// TIA Portal project "MQTT_Demo_V14" (V14)

(* hardware
DEVICE "S7-1200 station_1"  S7-1200 Station
   slot 0: "Rack_0"  Rack  V1.0
   slot 1: "MQTT_Demo"  CPU 1214C AC/DC/Rly  6ES7 214-1BG40-0XB0  V4.2
*)

// ===== PLC "MQTT_Demo"  CPU 1214C AC/DC/Rly =====

VAR_GLOBAL   // PLC tag table "Default tag table"
   "Clock_Byte" AT %MB0 : Byte;
   "Clock_10Hz" AT %M0.0 : Bool;
   "Clock_5Hz" AT %M0.1 : Bool;
   "Clock_2.5Hz" AT %M0.2 : Bool;
   "Clock_2Hz" AT %M0.3 : Bool;
   "Clock_1.25Hz" AT %M0.4 : Bool;
   "Clock_1Hz" AT %M0.5 : Bool;
   "Clock_0.625Hz" AT %M0.6 : Bool;
   "Clock_0.5Hz" AT %M0.7 : Bool;
   "System_Byte" AT %MB1 : Byte;
   "FirstScan" AT %M1.0 : Bool;
   "DiagStatusUpdate" AT %M1.1 : Bool;
   "AlwaysTRUE" AT %M1.2 : Bool;
   "AlwaysFALSE" AT %M1.3 : Bool;
   "mwTemp" AT %MW20 : Word;
   "DI_Good" AT %I0.0 : Bool;
   "DI_Bad" AT %I0.1 : Bool;
   "DQ_Error" AT %Q0.1 : Bool;
   "DQ_Busy" AT %Q0.0 : Bool;
END_VAR

TYPE "udtError_MQTT"
   STRUCT
      ConSendErr : Bool;   // Connect send error
      ConSendTO : Bool;   // Connect send timeout
      ConAckRcvErr : Bool;   // Connack receive error
      ConAckTO : Bool;   // Connack timeout
      ConAckIncReply : Bool;   // Conack incorrect reply (header)
      ConAckIncLen : Bool;   // Conack incorrect remaining length
      ConAckUnacProt : Bool;   // Conack unacceptable protocol version (0x01)
      ConAckIdRej : Bool;   // Conack ID rejected (0x02)
      ConAckSerUn : Bool;   // Conack server unavailable (0x03)
      ConAckUserPass : Bool;   // Conack incorerct user/password (0x04)
      ConAckNotAut : Bool;   // Conack not authorized (0x05)
      ConAckUnknown : Bool;   // Conack unknow erro code (>0x05)
      PubSendErr : Bool;   // Publish send error
      PubSendTO : Bool;   // Publish send timeout
      PubAckRcvErr : Bool;   // Puback receive error
      PubAckTO : Bool;   // Puback receive timeout
      PubAckIncReply : Bool;   // Puback incorerct reply (header)
      PubAckIncLen : Bool;   // Puback incorrect remaining length
      PubAckPacketID : Bool;   // Puback incorrect Packet ID
      TcpErr : Bool;   // TCP connection failed
      TcpTO : Bool;   // TCP connection timeout
      QueueOverflow : Bool;   // Queue overlow
   END_STRUCT;
END_TYPE

DATA_BLOCK "dbMQTT_Queue"   // DB1
{ S7_Optimized_Access := 'TRUE' }
VERSION : 0.1
   VAR
      iIndexWrite : Int;   // Write index
      iIndexMax : Int;   // Max elements in the queue
      bErrorOverfill : Bool;   // Queue overfill error detected
      Element : Array[1..50] of Struct
         iStatus : Int;
         iQOS : Int;
         sTopic : String;
         sValue : String;
      END_STRUCT;
   END_VAR
BEGIN
END_DATA_BLOCK

DATA_BLOCK "fbInsMaster_IBM"   // DB2
{ S7_Optimized_Access := 'TRUE' }
VERSION : 0.1
// stored: InstanceOfName fbMaster_IBM
"fbMaster_IBM"
BEGIN
END_DATA_BLOCK

DATA_BLOCK "fbInsMaster_Adafruit"   // DB4
{ S7_Optimized_Access := 'TRUE' }
VERSION : 0.1
// stored: InstanceOfName fbMaster_Adafruit
"fbMaster_Adafruit"
BEGIN
END_DATA_BLOCK

DATA_BLOCK "dbMessages"   // DB5
{ S7_Optimized_Access := 'TRUE' }
VERSION : 0.1
   VAR
      sMessage : Array[1..50] of String;
   END_VAR
BEGIN
   sMessage[1] := 'Knock Knock. Who`s there? Ice cream! Ice cream who? Ice cream if you don`t let me in!';
   sMessage[2] := 'Knock Knock. Who`s there? Noah. Noah who? Noah way to open the door?';
   sMessage[3] := 'Knock Knock. Who`s there? Cows go. Cows go who? No, cows go moo!';
   sMessage[4] := 'Knock Knock. Who`s there? Hatch. Hatch who? Bless you and please cover your mouth next time.';
   sMessage[5] := 'Knock Knock. Who`s there? Boo. Boo who? Don`t cry, it`s just a joke.';
   sMessage[6] := 'Knock Knock. Who`s there? Venice. Venice who? Venice this door gonna open?';
   sMessage[7] := 'Knock Knock. Who`s there? Lettuce! Lettuce who? Lettuce in!';
   sMessage[8] := 'Knock Knock. Who`s there? Scold. Scold who? Scold outside-let me in!';
   sMessage[9] := 'Knock Knock. Who`s there? Needle. Needle who? Needle little help gettin` in the door.';
   sMessage[10] := 'Knock Knock. Who`s there? Nana. Nana who? Nana your business who`s there.';
   sMessage[11] := 'Knock Knock. Who`s there? Isabelle. Isabelle who? Isabelle working, or should I keep knocking?';
   sMessage[12] := 'Knock Knock. Who`s there? Claire. Claire who? Claire the way; I`m coming in!';
   sMessage[13] := 'Knock Knock. Who`s there? Ben. Ben who? Ben knocking for 20 minutes!';
   sMessage[14] := 'Knock Knock. Who`s there? Tuna! Tuna who? Tuna piano and it`ll sound better!';
   sMessage[15] := 'Knock Knock. Who`s there? Snow! Snow who? Snow use, I`ve forgotten my key again!';
END_DATA_BLOCK

// folder: System blocks/Program resources

DATA_BLOCK "dbTCON_Adafruit"   // DB3
{ S7_Optimized_Access := 'TRUE' }
AUTHOR : SIMATIC
FAMILY : MC7Plus
NAME : TCON_Prm
VERSION : 1.0
// stored: InstanceOfName TCON_Param
"TCON_Param"
BEGIN
   ID := 1;
   REM_TSAP_ID[1] := B#16#07;
   REM_TSAP_ID[2] := B#16#5B;
   REM_STADDR[1] := 52;
   REM_STADDR[2] := 70;
   REM_STADDR[3] := 203;
   REM_STADDR[4] := 194;
END_DATA_BLOCK

DATA_BLOCK "dbTCON_IBM"   // DB6
{ S7_Optimized_Access := 'TRUE' }
AUTHOR : SIMATIC
FAMILY : MC7Plus
NAME : TCON_Prm
VERSION : 1.0
// stored: InstanceOfName TCON_Param
"TCON_Param"
BEGIN
   ID := 1;
   REM_TSAP_ID[1] := B#16#07;
   REM_TSAP_ID[2] := B#16#5B;
   REM_STADDR[1] := 169;
   REM_STADDR[2] := 45;
   REM_STADDR[3] := 2;
   REM_STADDR[4] := 20;
END_DATA_BLOCK

// folder: (top level)

FUNCTION_BLOCK "fbMQTT"   // FB1, SCL
{ S7_Optimized_Access := 'FALSE' }
VERSION : 0.1
   VAR_INPUT
      iInQueueSize : Int;
      sInClientID : String;   // Client ID, 23 char max
      sInUserName : String;
      sInPassword : String;
      bInCleanSession : Bool;   // 0=Reuse prev session; 1=Discard prev sessions and start new one
      bInResetError : Bool;
   END_VAR
   VAR_OUTPUT
      bOutError : Bool;
      bOutBusy : Bool;
      bOutTCPConnected : Bool;
      bOutMQTT_Connected : Bool;
      ERROR_MQTT : "udtError_MQTT";
   END_VAR
   VAR_IN_OUT
      TCON_Param : TCON_Param;
   END_VAR
   VAR
      fbTCON : TCON;
      fbTDISCON : TDISCON;
      fbTSEND : TSEND;
      fbTRCV : TRCV;
      TON_Timeout : TON_TIME;
      byData : Array[1..1000] of Byte;   // Max: id+user+password+buffer
      bTCP_Connected : Bool;
      bMQTT_Connected : Bool;
      bPubInProgress : Bool;
      iState : Int;   // Main state machine state
      iStatePrev : Int;   // Previous state
      iSelQueueIndex : Int;   // Selected queue index
      uiSendLen : UInt;   // Sending length
      udiReceiveLen : UDInt;
      uiPacketID : UInt := 1;
   END_VAR
   VAR_TEMP
      i : Int;
      iIndex : Int;
      iLen : Int;
      byTemp : Byte;
      uiTemp : UInt;
      bStateTransition : Bool;   // Transitioning between states
   END_VAR
   VAR CONSTANT
      ciStatusDisable : Int;   // Not ready
      ciStatusReady : Int := 10;   // Ready to be send to the server
      ciStateIDLE : Int := 0;
      ciStateCon : Int := 10;   // Connect
      ciStateConSend : Int := 15;
      ciStateConAck : Int := 20;
      ciStatePub : Int := 30;   // Publish
      ciStatePubSend : Int := 35;
      ciStatePubAck : Int := 40;
      ciStateEstablishTCP : Int := 50;   // Establish TCP connection
      ciStateError : Int := 60;
      ciStateRestart : Int := 70;
   END_VAR
BEGIN
   // Main state machine - case structure
   #iStatePrev := #iState;
   CASE #iState OF
           //**********************************************************************************************************************
       #ciStateIDLE: 
           // Update max queue index
           "dbMQTT_Queue".iIndexMax := #iInQueueSize;

           // Already select element to send?
           IF #iSelQueueIndex > 0 THEN
               IF #bTCP_Connected THEN
                   IF #bMQTT_Connected THEN
                       // MQTT is conencted - just publish new message
                       #iState := #ciStatePub;
                   ELSE
                       // MQTT connection is not established - sene conn message
                       #iState := #ciStateCon;
                   END_IF;
               ELSE
                   // TCP is not connected - try to establish the connection
                   #iState := #ciStateEstablishTCP;
               END_IF;
           ELSE
               // Find element in the queue to send
               FOR #i := 1 TO "dbMQTT_Queue".iIndexMax DO
                   // Check if element is ready in the queue
                   IF ("dbMQTT_Queue".Element[#i].iStatus = #ciStatusReady) THEN
                       #iSelQueueIndex := #i;
                       EXIT;
                   END_IF;
               END_FOR;
           END_IF;

           //**********************************************************************************************************************
       #ciStateCon: // Send connect message
           ////////////////////////////////////
           // Create connect message
           ////////////////////////////////////

           //********* Configure Fixed Header ***********//
           #iIndex := 1;
           #byData[#iIndex] := 2#00010000;   // Packet type 0x1; Flags 0x0 (reserved)
           #iIndex := #iIndex + 1;

           // Calculate remaining length (see MQTT doc)
           #iLen := 12 + LEN(#sInClientID);
           IF LEN(#sInUserName) > 0 THEN
               #iLen := #iLen + LEN(#sInUserName) + 2;
           END_IF;
           IF LEN(#sInPassword) > 0 THEN
               #iLen := #iLen + LEN(#sInPassword) + 2;
           END_IF;
           REPEAT
               #byTemp := INT_TO_BYTE(#iLen MOD 128);
               #iLen := #iLen / 128;
               // if there are more data to encode, set the top bit of this byte 286
               IF #iLen > 0 THEN
                   #byTemp := #byTemp OR 128;
               END_IF;
               #byData[#iIndex] := #byTemp;
               #iIndex := #iIndex + 1;
           UNTIL #iLen <= 0 END_REPEAT;

           //********* Variable Header ***********//
           #byData[#iIndex] := 16#00;    // Length MSB
           #iIndex := #iIndex + 1;
           #byData[#iIndex] := 16#04;    // Length LSB
           #iIndex := #iIndex + 1;
           #byData[#iIndex] := CHAR_TO_BYTE('M');
           #iIndex := #iIndex + 1;
           #byData[#iIndex] := CHAR_TO_BYTE('Q');
           #iIndex := #iIndex + 1;
           #byData[#iIndex] := CHAR_TO_BYTE('T');
           #iIndex := #iIndex + 1;
           #byData[#iIndex] := CHAR_TO_BYTE('T');
           #iIndex := #iIndex + 1;
           #byData[#iIndex] := 16#04;     // Protocol level 0x04
           #iIndex := #iIndex + 1;

           // Build connect flags, ignoring will message
           #byData[#iIndex] := 16#00;
           IF LEN(#sInUserName) > 0 THEN
               #byData[#iIndex] := #byData[#iIndex] OR 2#10000000;
           END_IF;
           IF LEN(#sInPassword) > 0 THEN
               #byData[#iIndex] := #byData[#iIndex] OR 2#01000000;
           END_IF;
           IF #bInCleanSession THEN
               #byData[#iIndex] := #byData[#iIndex] OR 2#00000010;
           END_IF;
           #iIndex := #iIndex + 1;
           #byData[#iIndex] := 16#0E;  // Keepalive MSB, in seconds
           #iIndex := #iIndex + 1;
           #byData[#iIndex] := 16#10;  // Keepalive LSB, in seconds
           #iIndex := #iIndex + 1;

           // Payload - client ID
           #iLen := LEN(#sInClientID);
           #byData[#iIndex] := WORD_TO_BYTE(SHR(IN := INT_TO_WORD(#iLen), N := 8));   // String lenght MSB
           #iIndex := #iIndex + 1;
           #byData[#iIndex] := WORD_TO_BYTE(INT_TO_WORD(#iLen) AND 16#00FF);   // String lenght LSB            
           #iIndex := #iIndex + 1;
           FOR #i := 1 TO #iLen DO
               #byData[#iIndex] := CHAR_TO_BYTE(#sInClientID[#i]);
               #iIndex := #iIndex + 1;
           END_FOR;

           // Payload - User name
           IF LEN(#sInUserName) > 0 THEN
               #iLen := LEN(#sInUserName);
               #byData[#iIndex] := WORD_TO_BYTE(SHR(IN := INT_TO_WORD(#iLen), N := 8));   // String lenght MSB
               #iIndex := #iIndex + 1;
               #byData[#iIndex] := WORD_TO_BYTE(INT_TO_WORD(#iLen) AND 16#00FF);   // String lenght LSB            
               #iIndex := #iIndex + 1;
               FOR #i := 1 TO #iLen DO
                   #byData[#iIndex] := CHAR_TO_BYTE(#sInUserName[#i]);
                   #iIndex := #iIndex + 1;
               END_FOR;
           END_IF;

           // Payload - password
           IF LEN(#sInPassword) > 0 THEN
               #iLen := LEN(#sInPassword);
               #byData[#iIndex] := WORD_TO_BYTE(SHR(IN := INT_TO_WORD(#iLen), N := 8));   // String lenght MSB
               #iIndex := #iIndex + 1;
               #byData[#iIndex] := WORD_TO_BYTE(INT_TO_WORD(#iLen) AND 16#00FF);   // String lenght LSB            
               #iIndex := #iIndex + 1;
               FOR #i := 1 TO #iLen DO
                   #byData[#iIndex] := CHAR_TO_BYTE(#sInPassword[#i]);
                   #iIndex := #iIndex + 1;
               END_FOR;
           END_IF;

           //********* Send Packet ***********//
           #uiSendLen := INT_TO_UINT(#iIndex - 1);   // Update packet length
           #iState := #ciStateConSend;  // Send packet packet    

           //**********************************************************************************************************************
       #ciStateConSend:
           IF #fbTSEND.DONE THEN
               // All good. Receive conack message
               // We know exactly the conack message size
               #udiReceiveLen := 4;
               #iState := #ciStateConAck;
           ELSIF #fbTSEND.ERROR THEN
               // Sending error
               #ERROR_MQTT.ConSendErr := true;
               #iState := #ciStateError;
           ELSIF #TON_Timeout.Q THEN
               #ERROR_MQTT.ConSendTO := true;
               #iState := #ciStateError;
           END_IF;

           //**********************************************************************************************************************
       #ciStateConAck:
           IF #fbTRCV.NDR THEN
               // Parse received data
               // We know that we got an expected length
               // Header should be 0x20
               IF #byData[1] <> 16#20 THEN
                   #ERROR_MQTT.ConAckIncReply := true;
                   #iState := #ciStateError;
               // Remaining lenght should be 2
               ELSIF #byData[2] <> 2 THEN
                   #ERROR_MQTT.ConAckIncLen := true;
                   #iState := #ciStateError;
               // TODO: Parse SP flag?
               // Return code should be 0    
               ELSIF #byData[4] <> 0 THEN
                   // Parse error code
                   IF #byData[4] = 1 THEN
                       #ERROR_MQTT.ConAckUnacProt := TRUE;
                   ELSIF #byData[4] = 2 THEN
                       #ERROR_MQTT.ConAckIdRej := TRUE;
                   ELSIF #byData[4] = 3 THEN
                       #ERROR_MQTT.ConAckSerUn := TRUE;
                   ELSIF #byData[4] = 4 THEN
                       #ERROR_MQTT.ConAckUserPass := TRUE;
                   ELSIF #byData[4] = 5 THEN
                       #ERROR_MQTT.ConAckNotAut := TRUE;
                   ELSE
                       #ERROR_MQTT.ConAckUnknown := TRUE;
                   END_IF;
                   #iState := #ciStateError;
               ELSE
                   // All good
                   #bMQTT_Connected := true;
                   #iState := #ciStatePub;
               END_IF;
           ELSIF #fbTRCV.ERROR THEN
               // Receive error
               #ERROR_MQTT.ConAckRcvErr := true;
               #iState := #ciStateError;
           ELSIF #TON_Timeout.Q THEN
               #ERROR_MQTT.ConAckTO := true;
               #iState := #ciStateError;
           END_IF;

           //**********************************************************************************************************************
       #ciStatePub:
           ////////////////////////////////////
           // Create publish message
           ////////////////////////////////////

           //********* Configure Fixed Header ***********//
           #iIndex := 1;
           #byData[#iIndex] := 2#00110000;   // Packet type 0x3;
           IF #bPubInProgress THEN
               #byData[#iIndex] := #byData[#iIndex] OR 2#00001000; // DUP flag. Re-delivery attempt
           ELSE
               // New send attempt - Increment Packet ID
               #uiPacketID := #uiPacketID + 1;
           END_IF;
           // QoS flag, assuming 0 by default
           IF "dbMQTT_Queue".Element[#iSelQueueIndex].iQOS = 1 THEN
               #byData[#iIndex] := #byData[#iIndex] OR 2#00000010; // QoS flag
           END_IF;
           //TODO: QoS 2 is not currently implemented by adafruit
           // TODO: Ignoring retain flag for now
           #iIndex := #iIndex + 1;

           // Calculate remaining length (see MQTT doc)
           // No lenght for the payload
           #iLen := LEN("dbMQTT_Queue".Element[#iSelQueueIndex].sTopic) + 2 + LEN("dbMQTT_Queue".Element[#iSelQueueIndex].sValue);
           IF "dbMQTT_Queue".Element[#iSelQueueIndex].iQOS > 0 THEN
               // Adding packet ID for QoS 1 and 2
               #iLen := #iLen + 2;
           END_IF;
           REPEAT
               #byTemp := INT_TO_BYTE(#iLen MOD 128);
               #iLen := #iLen / 128;
               // if there are more data to encode, set the top bit of this byte 286
               IF #iLen > 0 THEN
                   #byTemp := #byTemp OR 128;
               END_IF;
               #byData[#iIndex] := #byTemp;
               #iIndex := #iIndex + 1;
           UNTIL #iLen <= 0 END_REPEAT;

           //********* Variable Header ***********//
           // Topic name
           #iLen := LEN("dbMQTT_Queue".Element[#iSelQueueIndex].sTopic);
           #byData[#iIndex] := WORD_TO_BYTE(SHR(IN:=INT_TO_WORD(#iLen), N:=8));   // String lenght MSB
           #iIndex := #iIndex + 1;
           #byData[#iIndex] := WORD_TO_BYTE(INT_TO_WORD(#iLen) AND 16#00FF);   // String lenght LSB
           #iIndex := #iIndex + 1;
           FOR #i := 1 TO #iLen DO
               #byData[#iIndex] := CHAR_TO_BYTE("dbMQTT_Queue".Element[#iSelQueueIndex].sTopic[#i]);
               #iIndex := #iIndex + 1;
           END_FOR;
           // packet ID
           IF "dbMQTT_Queue".Element[#iSelQueueIndex].iQOS > 0 THEN
               #byData[#iIndex] := WORD_TO_BYTE(SHR(IN:=UINT_TO_WORD(#uiPacketID), N:=8));   // Packet ID MSB
               #iIndex := #iIndex + 1;
               #byData[#iIndex] := WORD_TO_BYTE(UINT_TO_WORD(#uiPacketID) AND 16#00FF);   // PacketID LSB
               #iIndex := #iIndex + 1;
           END_IF;

           //********* Payload ***********//
           // The exact data format is not defined in the MQTT spec
           // Assuming strings, without string length
           // According to the spec, server should calcualte the lenght of the payload
           #iLen := LEN("dbMQTT_Queue".Element[#iSelQueueIndex].sValue);
           FOR #i := 1 TO #iLen DO
               #byData[#iIndex] := CHAR_TO_BYTE("dbMQTT_Queue".Element[#iSelQueueIndex].sValue[#i]);
               #iIndex := #iIndex + 1;
           END_FOR;

           // Send message
           #bPubInProgress := true;
           #uiSendLen := INT_TO_UINT(#iIndex - 1);   // Update packet length
           #iState := #ciStatePubSend;

           //**********************************************************************************************************************
       #ciStatePubSend:
           IF #fbTSEND.DONE THEN
               // QoS=1: Should receive puback message
               IF "dbMQTT_Queue".Element[#iSelQueueIndex].iQOS = 1 THEN
                   #udiReceiveLen := 4;    // Wes should receive exactly 4 bytes
                   #iState := #ciStatePubAck;
               ELSE
                   // QoS=0; No response from the server
                   // Remove message from the queue
                   "dbMQTT_Queue".Element[#iSelQueueIndex].iStatus := #ciStatusDisable;
                   #iSelQueueIndex := 0;
                   #bPubInProgress := false;
                   #iState := #ciStateIDLE;
               END_IF;
               // TODO: Handle QoS 2?
           ELSIF #fbTSEND.ERROR THEN
               // Send error
               #ERROR_MQTT.PubSendErr := true;
               #iState := #ciStateError;
           ELSIF #TON_Timeout.Q THEN
               #ERROR_MQTT.PubSendTO := true;
               #iState := #ciStateError;
           END_IF;

           //**********************************************************************************************************************
       #ciStatePubAck:
           IF #fbTRCV.NDR THEN
               // Parse received data
               // We know that we got an expected length
               // Header should be 0x40
               IF #byData[1] <> 16#40 THEN
                   // Wrong pub ack header
                   #ERROR_MQTT.PubAckIncReply := TRUE;
                   #iState := #ciStateError;
               // Remaining length should be 2
               ELSIF #byData[2] <> 16#02 THEN
                   // Wrong pub ack remaining lenght
                   #ERROR_MQTT.PubAckIncLen := TRUE;
                   #iState := #ciStateError;
               ELSE
                   // Variable header = message id
                   #uiTemp := WORD_TO_UINT(SHL(IN := BYTE_TO_WORD(#byData[3]), N := 8) + BYTE_TO_WORD(#byData[4]));
                   IF #uiTemp <> #uiPacketID THEN
                       // Incorerct packet ID
                       #ERROR_MQTT.PubAckPacketID := TRUE;
                       #iState := #ciStateError;
                   ELSE
                       // All good. Reset queue and restart
                       "dbMQTT_Queue".Element[#iSelQueueIndex].iStatus := #ciStatusDisable;
                       #iSelQueueIndex := 0;
                       #bPubInProgress := false;
                       #iState := #ciStateIDLE;
                   END_IF;
               END_IF;
           ELSIF #fbTRCV.ERROR THEN
               // Receive error
               #ERROR_MQTT.PubAckRcvErr := TRUE;
               #iState := #ciStateError;
           ELSIF #TON_Timeout.Q THEN
               #ERROR_MQTT.PubAckTO := true;
               #iState := #ciStateError;
           END_IF;

           //**********************************************************************************************************************        
       #ciStateEstablishTCP:
           // Wait for done or error flag
           IF #fbTCON.DONE THEN
               // TCP connection established 
               #bTCP_Connected := true;
               #bMQTT_Connected := false;
               #iState := #ciStateCon;
           ELSIF #fbTCON.ERROR THEN
               // Connection failed
               #ERROR_MQTT.TcpErr := true;
               #iState := #ciStateError;
           ELSIF #TON_Timeout.Q THEN
               #ERROR_MQTT.TcpTO := true;
               #iState := #ciStateError;
           END_IF;

           //**********************************************************************************************************************
       #ciStateError:
           // Reset TCP connection
           #bMQTT_Connected := false;
           #bTCP_Connected := false;
           IF #fbTDISCON.DONE OR #fbTDISCON.ERROR THEN
               #iState := #ciStateRestart;
           ELSIF #TON_Timeout.Q THEN
               // Already wait for timeout, just jump to idle
               #iState := #ciStateIDLE;
           END_IF;

           //**********************************************************************************************************************
       #ciStateRestart:
           // Wait before restarting after the error
           IF #TON_Timeout.Q THEN
               // Restart from IDLE
               #iState := #ciStateIDLE;
           END_IF;

           //**********************************************************************************************************************
       ELSE    // Something is not right - reset state
           #iState := #ciStateIDLE;
   END_CASE;


   //**********************************************************************************************************************
   // Reset all errors
   IF #bInResetError THEN
       #ERROR_MQTT.ConSendErr := FALSE;
       #ERROR_MQTT.ConSendTO := FALSE;
       #ERROR_MQTT.ConAckRcvErr := FALSE;
       #ERROR_MQTT.ConAckTO := FALSE;
       #ERROR_MQTT.ConAckIncReply := FALSE;
       #ERROR_MQTT.ConAckIncLen := FALSE;
       #ERROR_MQTT.ConAckUnacProt := FALSE;
       #ERROR_MQTT.ConAckIdRej := FALSE;
       #ERROR_MQTT.ConAckSerUn := FALSE;
       #ERROR_MQTT.ConAckUserPass := FALSE;
       #ERROR_MQTT.ConAckNotAut := FALSE;
       #ERROR_MQTT.ConAckUnknown := FALSE;
       #ERROR_MQTT.PubSendErr := FALSE;
       #ERROR_MQTT.PubSendTO := FALSE;
       #ERROR_MQTT.PubAckRcvErr := FALSE;
       #ERROR_MQTT.PubAckTO := FALSE;
       #ERROR_MQTT.PubAckIncReply := FALSE;
       #ERROR_MQTT.PubAckIncLen := FALSE;
       #ERROR_MQTT.PubAckPacketID := FALSE;
       #ERROR_MQTT.TcpErr := FALSE;
       #ERROR_MQTT.TcpTO := FALSE;
       #ERROR_MQTT.QueueOverflow := FALSE;
   END_IF;

   // Queue overlow error
   IF "dbMQTT_Queue".bErrorOverfill THEN
       #ERROR_MQTT.QueueOverflow := TRUE;
       "dbMQTT_Queue".bErrorOverfill := FALSE;
   END_IF;

   // Timeoout timer
   #bStateTransition := #iState <> #iStatePrev;
   #TON_Timeout(IN := ((NOT #bStateTransition) AND (#iState <> #ciStateIDLE)), PT := T#20S);

   // At least one erorr is active - set output error flag
   #bOutError :=
       #ERROR_MQTT.ConSendErr OR
       #ERROR_MQTT.ConSendTO OR
       #ERROR_MQTT.ConAckRcvErr OR
       #ERROR_MQTT.ConAckTO OR
       #ERROR_MQTT.ConAckIncReply OR
       #ERROR_MQTT.ConAckIncLen OR
       #ERROR_MQTT.ConAckUnacProt OR
       #ERROR_MQTT.ConAckIdRej OR
       #ERROR_MQTT.ConAckSerUn OR
       #ERROR_MQTT.ConAckUserPass OR
       #ERROR_MQTT.ConAckNotAut OR
       #ERROR_MQTT.ConAckUnknown OR
       #ERROR_MQTT.PubSendErr OR
       #ERROR_MQTT.PubSendTO OR
       #ERROR_MQTT.PubAckRcvErr OR
       #ERROR_MQTT.PubAckTO OR
       #ERROR_MQTT.PubAckIncReply OR
       #ERROR_MQTT.PubAckIncLen OR
       #ERROR_MQTT.PubAckPacketID OR
       #ERROR_MQTT.TcpErr OR
       #ERROR_MQTT.TcpTO OR
       #ERROR_MQTT.QueueOverflow;

   // Block is busy output flag
   #bOutBusy := (#iState <> #ciStateIDLE) AND (NOT #bOutError);

   // TCP and MQTT conencted outputs
   #bOutTCPConnected := #bTCP_Connected;
   #bOutMQTT_Connected := #bMQTT_Connected;


   //**********************************************************************************************************************
   // Communicaiton FBs
   #fbTCON(REQ:= (#iState = #ciStateEstablishTCP),
           ID:= #TCON_Param.ID,
           CONNECT:=#TCON_Param);

   #fbTDISCON(REQ:=(#iState = #ciStateError),
              ID:=#TCON_Param.ID);

   #fbTSEND(REQ := (#iState = #ciStateConSend) OR (#iState = #ciStatePubSend),
            ID := #TCON_Param.ID,
            LEN := #uiSendLen,
            DATA := #byData);

   #fbTRCV(EN_R := (#iState = #ciStateConAck) OR (#iState = #ciStatePubAck),
           ID:=#TCON_Param.ID,
           LEN:=#udiReceiveLen,
           DATA:=#byData);

   ENO := TRUE;
END_FUNCTION_BLOCK

FUNCTION_BLOCK "fbMaster_Adafruit"   // FB2, LAD
TITLE = Master FB
{ S7_Optimized_Access := 'TRUE' }
VERSION : 0.1
   VAR
      FP_PartGood : Bool;
      FP_PartBad : Bool;
      bMachineRunning : Bool;
      bOneMinutePulse : Bool;   // One shot one minute pulse
      diPartsGoodTotal : DInt;
      diPartsBadTotal : DInt;
      diPartsTotal : DInt;
      diPartsGoodMinute : DInt;
      diPartsBadMinute : DInt;
      diPartsMinute : DInt;
      rRunTimeSec : Real;
      rAvailability : Real;
      rPerformance : Real;
      rQuality : Real;
      diQuality : DInt;
      rOEE : Real;
      diOEE_Per : DInt;   // OEE in percents
      diOEE_PerAvg : DInt;   // Average OEE in percent
      iMessageIndex : Int;
      AVG_OEE : "fbRunningAverage";
      TON_OneMinute : TON_TIME;
      MQTT_Main : "fbMQTT";
      TON_ResetError : TON_TIME;
      TOF_Busy : TOF_TIME;
      TOF_MachineRunning : TOF_TIME;
      TONR_MachineRunTime : TONR_TIME;
   END_VAR
   VAR_TEMP
      rTemp : Real;
      bBusy : Bool;
      bTCP_Connected : Bool;
      bMQTT_Connected : Bool;
   END_VAR
   VAR CONSTANT
      cdiPlannedPartPerMinute : DInt := 30;   // Parts per minute rate
      crPlannedTimeSecPerMin : Real := 60.0;   // Planned time in seconds per interval (minute)
   END_VAR
   VAR_TEMP   // added for the SCL form of the ladder/FBD networks
      _w1 : Bool;
      _w2 : Bool;
   END_VAR
BEGIN

REGION Network 1: Made Good or Bad part
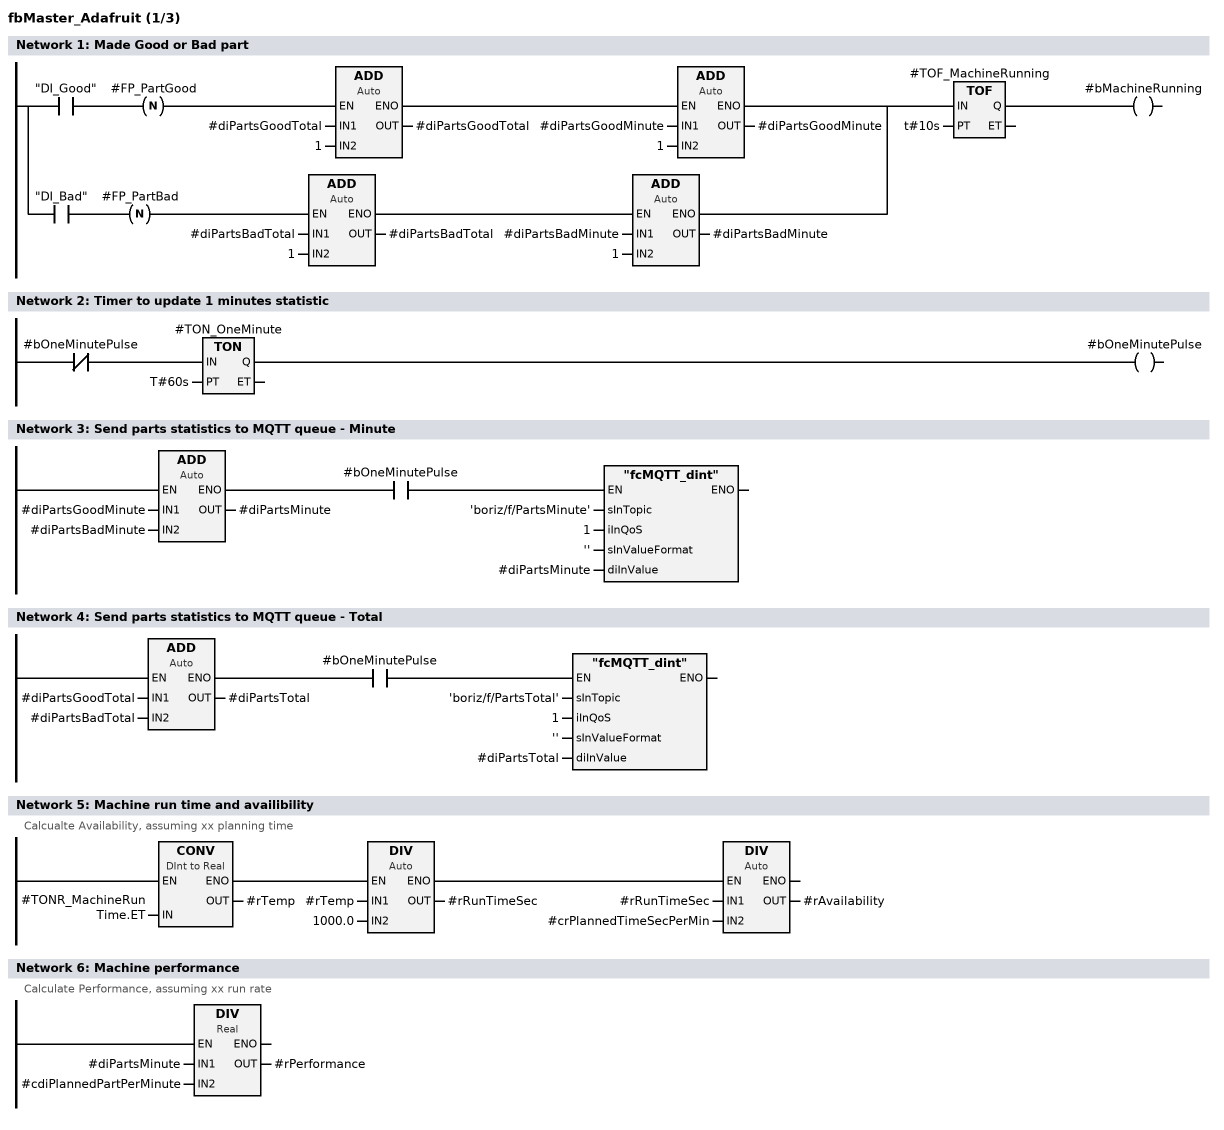
   #_w1 := NOT "DI_Good" AND #FP_PartGood;   // falling edge
   #FP_PartGood := "DI_Good";
   IF #_w1 THEN
       #diPartsGoodTotal := #diPartsGoodTotal + 1;
       #diPartsGoodMinute := #diPartsGoodMinute + 1;
   END_IF;
   #_w2 := NOT "DI_Bad" AND #FP_PartBad;   // falling edge
   #FP_PartBad := "DI_Bad";
   IF #_w2 THEN
       #diPartsBadTotal := #diPartsBadTotal + 1;
       #diPartsBadMinute := #diPartsBadMinute + 1;
   END_IF;
   #TOF_MachineRunning(IN := #_w1 OR #_w2, PT := t#10s);   // TOF
   #bMachineRunning := #TOF_MachineRunning.Q;
END_REGION

REGION Network 2: Timer to update 1 minutes statistic
   #TON_OneMinute(IN := NOT #bOneMinutePulse, PT := T#60s);   // TON
   #bOneMinutePulse := #TON_OneMinute.Q;
END_REGION

REGION Network 3: Send parts statistics to MQTT queue - Minute
   RUNG wire#powerrail
      Add(in1 := #diPartsGoodMinute, in2 := #diPartsBadMinute, out => #diPartsMinute)
      Contact( #bOneMinutePulse )
      "fcMQTT_dint"(sInTopic := 'boriz/f/PartsMinute', iInQoS := 1, sInValueFormat := '', diInValue := #diPartsMinute)
   END_RUNG
   // the same network as SCL:
   #diPartsMinute := #diPartsGoodMinute + #diPartsBadMinute;
   IF #bOneMinutePulse THEN
       "fcMQTT_dint"(sInTopic := 'boriz/f/PartsMinute',
                     iInQoS := 1,
                     sInValueFormat := '',
                     diInValue := #diPartsMinute);
   END_IF;
END_REGION

REGION Network 4: Send parts statistics to MQTT queue - Total
   RUNG wire#powerrail
      Add(in1 := #diPartsGoodTotal, in2 := #diPartsBadTotal, out => #diPartsTotal)
      Contact( #bOneMinutePulse )
      "fcMQTT_dint"(sInTopic := 'boriz/f/PartsTotal', iInQoS := 1, sInValueFormat := '', diInValue := #diPartsTotal)
   END_RUNG
   // the same network as SCL:
   #diPartsTotal := #diPartsGoodTotal + #diPartsBadTotal;
   IF #bOneMinutePulse THEN
       "fcMQTT_dint"(sInTopic := 'boriz/f/PartsTotal',
                     iInQoS := 1,
                     sInValueFormat := '',
                     diInValue := #diPartsTotal);
   END_IF;
END_REGION

REGION Network 5: Machine run time and availibility
   // Calcualte Availability, assuming xx planning time
   RUNG wire#powerrail
      { S7_Templates := "[SrcType := DInt, DestType := Real]" } Convert(in := #TONR_MachineRunTime.ET, out => #rTemp)
      Div(in1 := #rTemp, in2 := 1000.0, out => #rRunTimeSec)
      Div(in1 := #rRunTimeSec, in2 := #crPlannedTimeSecPerMin, out => #rAvailability)
   END_RUNG
   // the same network as SCL:
   #rTemp := DINT_TO_REAL(#TONR_MachineRunTime.ET);
   #rRunTimeSec := #rTemp / 1000.0;
   #rAvailability := #rRunTimeSec / #crPlannedTimeSecPerMin;
END_REGION

REGION Network 6: Machine performance
   // Calculate Performance, assuming xx run rate
   RUNG wire#powerrail
      { S7_Templates := "SrcType := Real" } Div(in1 := #diPartsMinute, in2 := #cdiPlannedPartPerMinute, out => #rPerformance)
   END_RUNG
   // the same network as SCL:
   #rPerformance := #diPartsMinute / #cdiPlannedPartPerMinute;
END_REGION

REGION Network 7: Machine quality
   // Calculate Quality
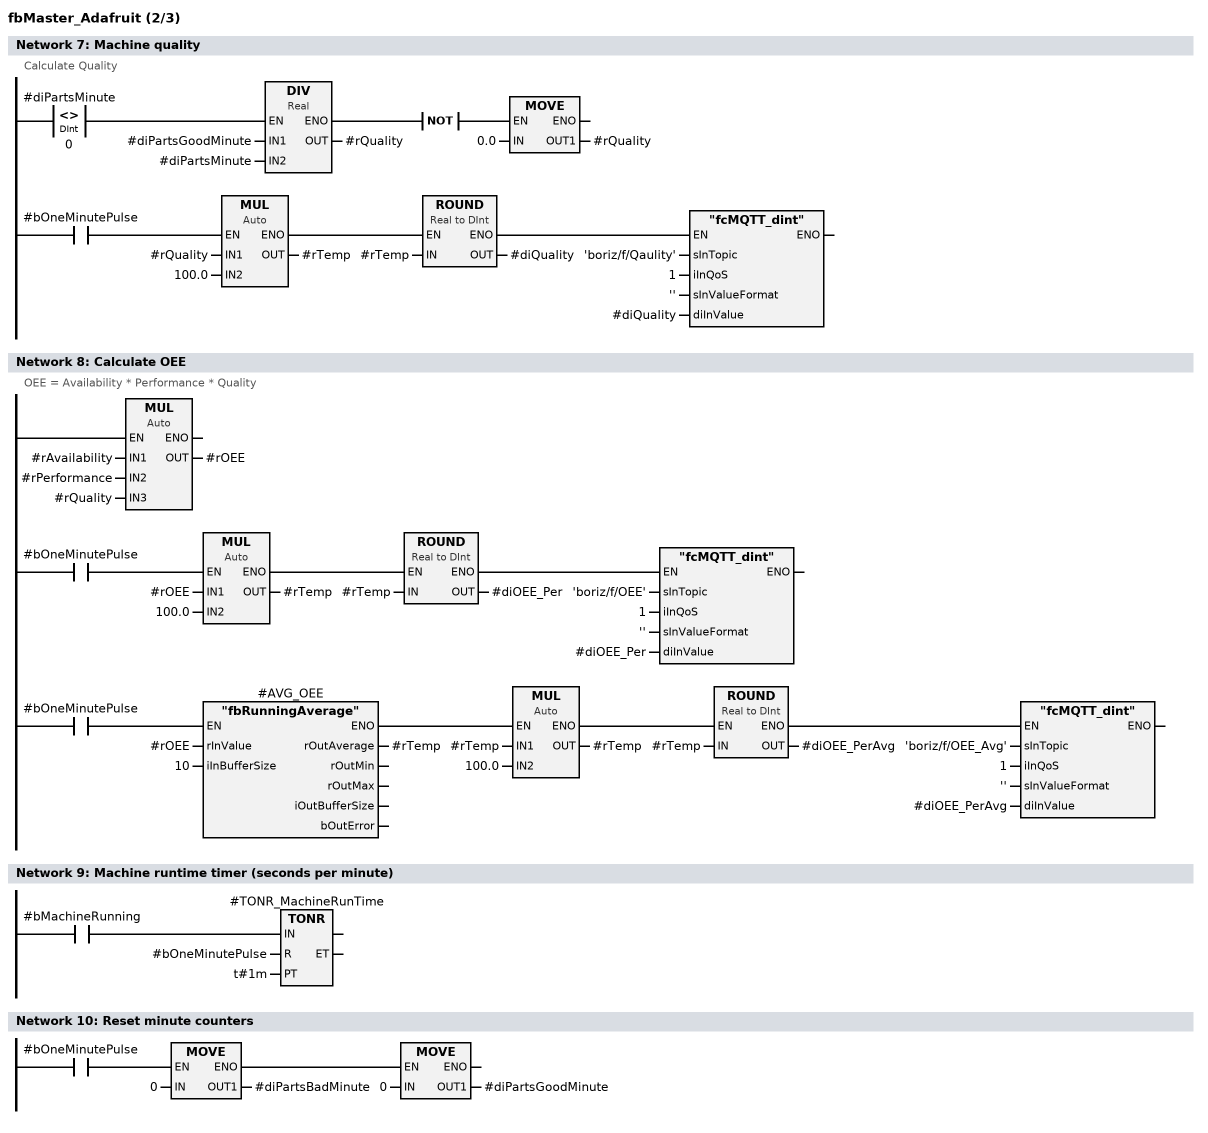
   RUNG wire#powerrail
      { S7_Templates := "SrcType := DInt" } NE_Contact(in1 := #diPartsMinute, in2 := 0)
      { S7_Templates := "SrcType := Real" } Div(in1 := #diPartsGoodMinute, in2 := #diPartsMinute, out => #rQuality)
      Not()
      Move(in := 0.0, out1 => #rQuality)
   END_RUNG
   RUNG wire#powerrail
      Contact( #bOneMinutePulse )
      Mul(in1 := #rQuality, in2 := 100.0, out => #rTemp)
      { S7_Templates := "[SrcType := Real, DestType := DInt]" } Round(in := #rTemp, out => #diQuality)
      "fcMQTT_dint"(sInTopic := 'boriz/f/Qaulity', iInQoS := 1, sInValueFormat := '', diInValue := #diQuality)
   END_RUNG
   // the same network as SCL:
   #_w1 := #diPartsMinute <> 0;
   IF #_w1 THEN #rQuality := #diPartsGoodMinute / #diPartsMinute; END_IF;
   IF NOT #_w1 THEN #rQuality := 0.0; END_IF;
   IF #bOneMinutePulse THEN
       #rTemp := #rQuality * 100.0;
       #diQuality := ROUND(#rTemp);
       "fcMQTT_dint"(sInTopic := 'boriz/f/Qaulity', iInQoS := 1, sInValueFormat := '', diInValue := #diQuality);
   END_IF;
END_REGION

REGION Network 8: Calculate OEE
   // OEE = Availability * Performance * Quality
   RUNG wire#powerrail
      Mul(in1 := #rAvailability, in2 := #rPerformance, in3 := #rQuality, out => #rOEE)
   END_RUNG
   RUNG wire#powerrail
      Contact( #bOneMinutePulse )
      Mul(in1 := #rOEE, in2 := 100.0, out => #rTemp)
      { S7_Templates := "[SrcType := Real, DestType := DInt]" } Round(in := #rTemp, out => #diOEE_Per)
      "fcMQTT_dint"(sInTopic := 'boriz/f/OEE', iInQoS := 1, sInValueFormat := '', diInValue := #diOEE_Per)
   END_RUNG
   RUNG wire#powerrail
      Contact( #bOneMinutePulse )
      #AVG_OEE(rInValue := #rOEE, iInBufferSize := 10, rOutAverage => #rTemp, rOutMin =>, rOutMax =>, iOutBufferSize =>, bOutError =>)
      Mul(in1 := #rTemp, in2 := 100.0, out => #rTemp)
      { S7_Templates := "[SrcType := Real, DestType := DInt]" } Round(in := #rTemp, out => #diOEE_PerAvg)
      "fcMQTT_dint"(sInTopic := 'boriz/f/OEE_Avg', iInQoS := 1, sInValueFormat := '', diInValue := #diOEE_PerAvg)
   END_RUNG
   // the same network as SCL:
   #rOEE := #rAvailability * #rPerformance * #rQuality;
   IF #bOneMinutePulse THEN
       #rTemp := #rOEE * 100.0;
       #diOEE_Per := ROUND(#rTemp);
       "fcMQTT_dint"(sInTopic := 'boriz/f/OEE', iInQoS := 1, sInValueFormat := '', diInValue := #diOEE_Per);
   END_IF;
   #AVG_OEE(EN := #bOneMinutePulse, rInValue := #rOEE, iInBufferSize := 10, rOutAverage => #rTemp, ENO => #_w1);   // "fbRunningAverage"
   IF #_w1 THEN
       #rTemp := #rTemp * 100.0;
       #diOEE_PerAvg := ROUND(#rTemp);
       "fcMQTT_dint"(sInTopic := 'boriz/f/OEE_Avg', iInQoS := 1, sInValueFormat := '', diInValue := #diOEE_PerAvg);
   END_IF;
END_REGION

REGION Network 9: Machine runtime timer (seconds per minute)
   #TONR_MachineRunTime(IN := #bMachineRunning, R := #bOneMinutePulse, PT := t#1m);   // TONR
END_REGION

REGION Network 10: Reset minute counters
   RUNG wire#powerrail
      Contact( #bOneMinutePulse )
      Move(in := 0, out1 => #diPartsBadMinute)
      Move(in := 0, out1 => #diPartsGoodMinute)
   END_RUNG
   // the same network as SCL:
   IF #bOneMinutePulse THEN
       #diPartsBadMinute := 0;
       #diPartsGoodMinute := 0;
   END_IF;
END_REGION

REGION Network 11: Send periodic message
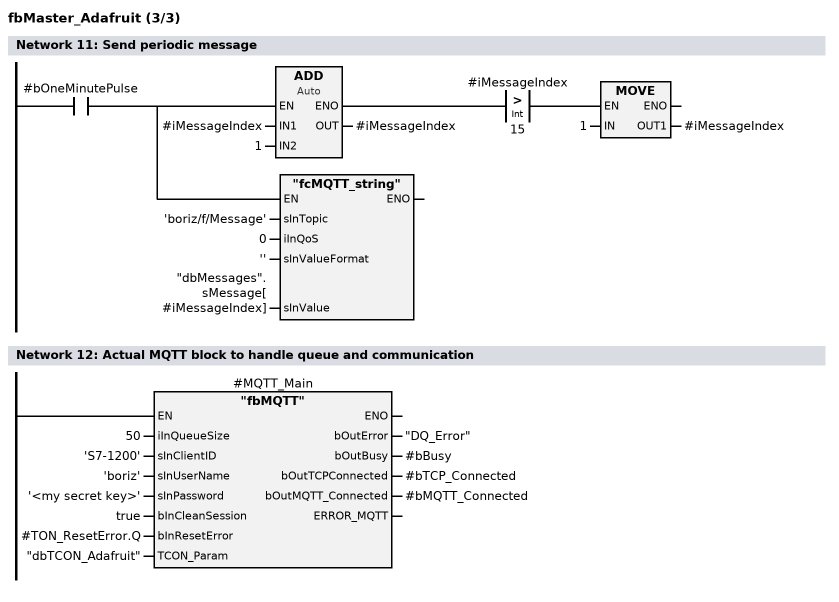
   RUNG wire#powerrail
      Contact( #bOneMinutePulse )
      wire#w1
      Add(in1 := #iMessageIndex, in2 := 1, out => #iMessageIndex)
      { S7_Templates := "SrcType := Int" } GT_Contact(in1 := #iMessageIndex, in2 := 15)
      Move(in := 1, out1 => #iMessageIndex)
   END_RUNG
   RUNG wire#w1
      "fcMQTT_string"(sInTopic := 'boriz/f/Message', iInQoS := 0, sInValueFormat := '', sInValue := "dbMessages".sMessage[#iMessageIndex])
   END_RUNG
   // the same network as SCL:
   IF #bOneMinutePulse THEN #iMessageIndex := #iMessageIndex + 1; END_IF;
   IF #bOneMinutePulse AND (#iMessageIndex > 15) THEN #iMessageIndex := 1; END_IF;
   IF #bOneMinutePulse THEN
       "fcMQTT_string"(sInTopic := 'boriz/f/Message',
                       iInQoS := 0,
                       sInValueFormat := '',
                       sInValue := "dbMessages".sMessage[#iMessageIndex]);
   END_IF;
END_REGION

REGION Network 12: Actual MQTT block to handle queue and communication
   RUNG wire#powerrail
      #MQTT_Main(iInQueueSize := 50, sInClientID := 'S7-1200', sInUserName := 'boriz', sInPassword := '<my secret key>', bInCleanSession := true, bInResetError := #TON_ResetError.Q, TCON_Param := "dbTCON_Adafruit", bOutError => "DQ_Error", bOutBusy => #bBusy, bOutTCPConnected => #bTCP_Connected, bOutMQTT_Connected => #bMQTT_Connected, ERROR_MQTT =>)
   END_RUNG
   // the same network as SCL:
   #MQTT_Main(iInQueueSize := 50,   // "fbMQTT"
              sInClientID := 'S7-1200',
              sInUserName := 'boriz',
              sInPassword := '<my secret key>',
              bInCleanSession := true,
              bInResetError := #TON_ResetError.Q,
              TCON_Param := "dbTCON_Adafruit",
              bOutError => "DQ_Error",
              bOutBusy => #bBusy,
              bOutTCPConnected => #bTCP_Connected,
              bOutMQTT_Connected => #bMQTT_Connected);
END_REGION
END_FUNCTION_BLOCK

FUNCTION_BLOCK "fbRunningAverage"   // FB3, SCL
{ S7_Optimized_Access := 'TRUE' }
VERSION : 0.1
   VAR_INPUT
      rInValue : Real;   // Input value
      iInBufferSize : Int;   // Requested buffer size
   END_VAR
   VAR_OUTPUT
      rOutAverage : Real;   // Average value
      rOutMin : Real;   // Minimum
      rOutMax : Real;   // Maximum
      iOutBufferSize : Real;   // Actual buffer size (limited to the size of the internal array)
      bOutError : Bool;   // Error - requested buffer size is greater than intrnal array size
   END_VAR
   VAR
      ValueHistory : Array[1..120] of Real;
   END_VAR
   VAR_TEMP
      iBufferSize : Int;
      i : Int;
      rSum : Real;
      rMin : Real;
      rMax : Real;
   END_VAR
   VAR CONSTANT
      ciValueHistorySize : Int := 120;
   END_VAR
BEGIN
       // Shift history array left by 1
       UMOVE_BLK(IN:=#ValueHistory[1], COUNT:=INT_TO_UDINT(#ciValueHistorySize - 1), OUT=>#ValueHistory[2]);

       // Add new value
       #ValueHistory[1] := #rInValue;

       IF #iInBufferSize > 1 THEN

           // Limit buffer size to the size of the array
           IF #iInBufferSize <= #ciValueHistorySize THEN
               #iBufferSize := #iInBufferSize;
               #bOutError := false;
           ELSE
               #iBufferSize := #ciValueHistorySize;
               #bOutError := true;
           END_IF;

           // Cycle throough the array
           #rSum := 0.0;
           #rMax := -3.402822E+38;
           #rMin := 3.402822E+38;
           FOR #i := 1 TO #iBufferSize BY 1 DO

               // Min/max logic
               IF #ValueHistory[#i] > #rMax THEN
                   #rMax := #ValueHistory[#i];
               END_IF;
               IF #ValueHistory[#i] < #rMin THEN
                   #rMin := #ValueHistory[#i];
               END_IF;

               // Calcualte sum
               #rSum := #rSum + #ValueHistory[#i];
           END_FOR;

           // Calculate average
           #rOutAverage := #rSum / (DINT_TO_REAL(#iBufferSize));
           #rOutMin := #rMin;
           #rOutMax := #rMax;
       ELSE
           // Buffer size is 1 - no averaging
           #iOutBufferSize := 1;
           #rOutAverage := #rInValue;
           #rOutMin := #rInValue;
           #rOutMax := #rInValue;
       END_IF;

       // Output actual buffer size
       #iOutBufferSize := #iBufferSize;

       ENO := TRUE;
END_FUNCTION_BLOCK

FUNCTION_BLOCK "fbMaster_IBM"   // FB4, LAD
TITLE = Master FB
{ S7_Optimized_Access := 'TRUE' }
VERSION : 0.1
   VAR
      FP_PartGood : Bool;
      FP_PartBad : Bool;
      bMachineRunning : Bool;
      bOneMinutePulse : Bool;   // One shot one minute pulse
      diPartsGoodTotal : DInt;
      diPartsBadTotal : DInt;
      diPartsTotal : DInt;
      diPartsGoodMinute : DInt;
      diPartsBadMinute : DInt;
      diPartsMinute : DInt;
      rRunTimeSec : Real;
      rAvailability : Real;
      rPerformance : Real;
      rQuality : Real;
      diQuality : DInt;
      rOEE : Real;
      diOEE_Per : DInt;   // OEE in percents
      diOEE_PerAvg : DInt;   // Average OEE in percent
      iMessageIndex : Int;
      AVG_OEE : "fbRunningAverage";
      TON_OneMinute : TON_TIME;
      MQTT_Main : "fbMQTT";
      TON_ResetError : TON_TIME;
      TOF_Busy : TOF_TIME;
      TOF_MachineRunning : TOF_TIME;
      TONR_MachineRunTime : TONR_TIME;
   END_VAR
   VAR_TEMP
      rTemp : Real;
      bBusy : Bool;
      bTCP_Connected : Bool;
      bMQTT_Connected : Bool;
   END_VAR
   VAR CONSTANT
      cdiPlannedPartPerMinute : DInt := 30;   // Parts per minute rate
      crPlannedTimeSecPerMin : Real := 60.0;   // Planned time in seconds per interval (minute)
   END_VAR
   VAR_TEMP   // added for the SCL form of the ladder/FBD networks
      _w1 : Bool;
      _w2 : Bool;
   END_VAR
BEGIN

REGION Network 1: Made Good or Bad part
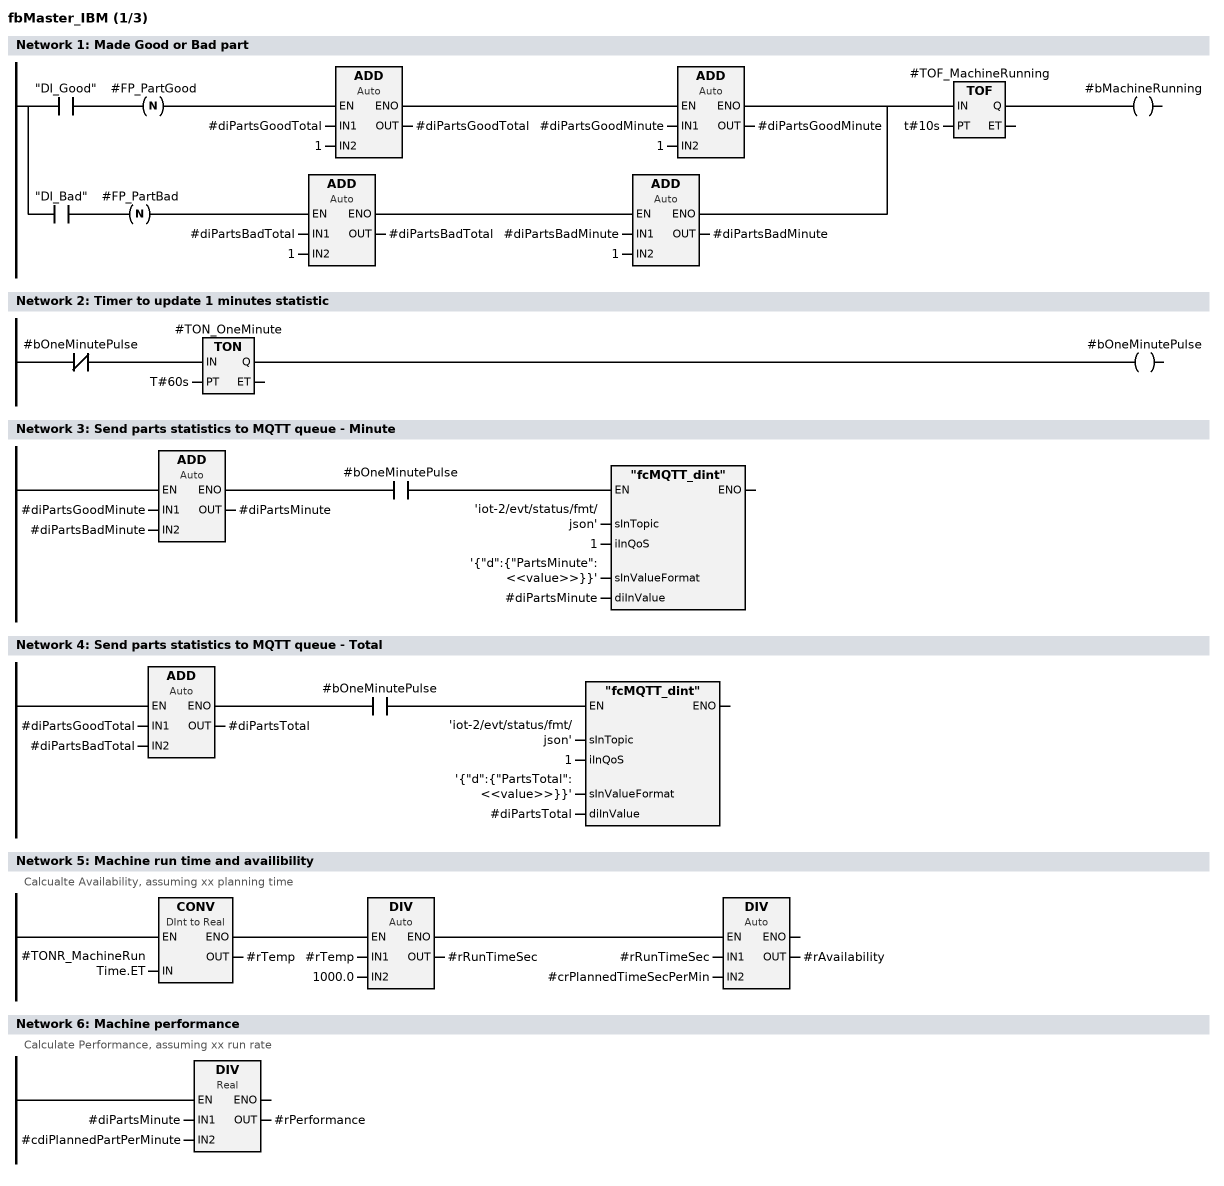
   #_w1 := NOT "DI_Good" AND #FP_PartGood;   // falling edge
   #FP_PartGood := "DI_Good";
   IF #_w1 THEN
       #diPartsGoodTotal := #diPartsGoodTotal + 1;
       #diPartsGoodMinute := #diPartsGoodMinute + 1;
   END_IF;
   #_w2 := NOT "DI_Bad" AND #FP_PartBad;   // falling edge
   #FP_PartBad := "DI_Bad";
   IF #_w2 THEN
       #diPartsBadTotal := #diPartsBadTotal + 1;
       #diPartsBadMinute := #diPartsBadMinute + 1;
   END_IF;
   #TOF_MachineRunning(IN := #_w1 OR #_w2, PT := t#10s);   // TOF
   #bMachineRunning := #TOF_MachineRunning.Q;
END_REGION

REGION Network 2: Timer to update 1 minutes statistic
   #TON_OneMinute(IN := NOT #bOneMinutePulse, PT := T#60s);   // TON
   #bOneMinutePulse := #TON_OneMinute.Q;
END_REGION

REGION Network 3: Send parts statistics to MQTT queue - Minute
   RUNG wire#powerrail
      Add(in1 := #diPartsGoodMinute, in2 := #diPartsBadMinute, out => #diPartsMinute)
      Contact( #bOneMinutePulse )
      "fcMQTT_dint"(sInTopic := 'iot-2/evt/status/fmt/json', iInQoS := 1, sInValueFormat := '{"d":{"PartsMinute":<<value>>}}', diInValue := #diPartsMinute)
   END_RUNG
   // the same network as SCL:
   #diPartsMinute := #diPartsGoodMinute + #diPartsBadMinute;
   IF #bOneMinutePulse THEN
       "fcMQTT_dint"(sInTopic := 'iot-2/evt/status/fmt/json',
                     iInQoS := 1,
                     sInValueFormat := '{"d":{"PartsMinute":<<value>>}}',
                     diInValue := #diPartsMinute);
   END_IF;
END_REGION

REGION Network 4: Send parts statistics to MQTT queue - Total
   RUNG wire#powerrail
      Add(in1 := #diPartsGoodTotal, in2 := #diPartsBadTotal, out => #diPartsTotal)
      Contact( #bOneMinutePulse )
      "fcMQTT_dint"(sInTopic := 'iot-2/evt/status/fmt/json', iInQoS := 1, sInValueFormat := '{"d":{"PartsTotal":<<value>>}}', diInValue := #diPartsTotal)
   END_RUNG
   // the same network as SCL:
   #diPartsTotal := #diPartsGoodTotal + #diPartsBadTotal;
   IF #bOneMinutePulse THEN
       "fcMQTT_dint"(sInTopic := 'iot-2/evt/status/fmt/json',
                     iInQoS := 1,
                     sInValueFormat := '{"d":{"PartsTotal":<<value>>}}',
                     diInValue := #diPartsTotal);
   END_IF;
END_REGION

REGION Network 5: Machine run time and availibility
   // Calcualte Availability, assuming xx planning time
   RUNG wire#powerrail
      { S7_Templates := "[SrcType := DInt, DestType := Real]" } Convert(in := #TONR_MachineRunTime.ET, out => #rTemp)
      Div(in1 := #rTemp, in2 := 1000.0, out => #rRunTimeSec)
      Div(in1 := #rRunTimeSec, in2 := #crPlannedTimeSecPerMin, out => #rAvailability)
   END_RUNG
   // the same network as SCL:
   #rTemp := DINT_TO_REAL(#TONR_MachineRunTime.ET);
   #rRunTimeSec := #rTemp / 1000.0;
   #rAvailability := #rRunTimeSec / #crPlannedTimeSecPerMin;
END_REGION

REGION Network 6: Machine performance
   // Calculate Performance, assuming xx run rate
   RUNG wire#powerrail
      { S7_Templates := "SrcType := Real" } Div(in1 := #diPartsMinute, in2 := #cdiPlannedPartPerMinute, out => #rPerformance)
   END_RUNG
   // the same network as SCL:
   #rPerformance := #diPartsMinute / #cdiPlannedPartPerMinute;
END_REGION

REGION Network 7: Machine quality
   // Calculate Quality
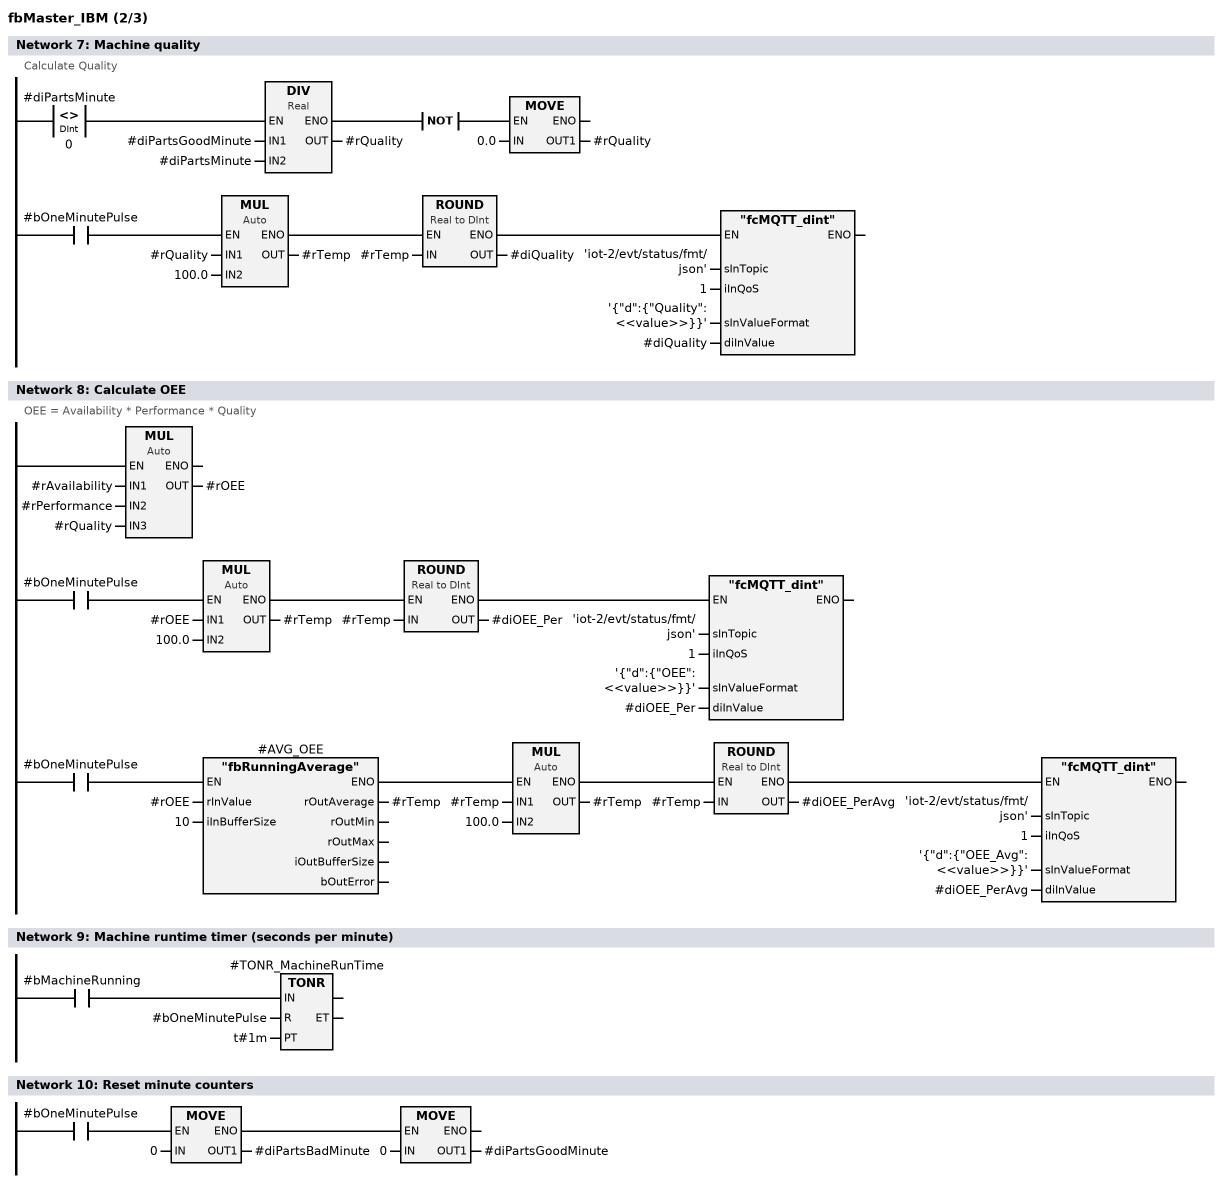
   RUNG wire#powerrail
      { S7_Templates := "SrcType := DInt" } NE_Contact(in1 := #diPartsMinute, in2 := 0)
      { S7_Templates := "SrcType := Real" } Div(in1 := #diPartsGoodMinute, in2 := #diPartsMinute, out => #rQuality)
      Not()
      Move(in := 0.0, out1 => #rQuality)
   END_RUNG
   RUNG wire#powerrail
      Contact( #bOneMinutePulse )
      Mul(in1 := #rQuality, in2 := 100.0, out => #rTemp)
      { S7_Templates := "[SrcType := Real, DestType := DInt]" } Round(in := #rTemp, out => #diQuality)
      "fcMQTT_dint"(sInTopic := 'iot-2/evt/status/fmt/json', iInQoS := 1, sInValueFormat := '{"d":{"Quality":<<value>>}}', diInValue := #diQuality)
   END_RUNG
   // the same network as SCL:
   #_w1 := #diPartsMinute <> 0;
   IF #_w1 THEN #rQuality := #diPartsGoodMinute / #diPartsMinute; END_IF;
   IF NOT #_w1 THEN #rQuality := 0.0; END_IF;
   IF #bOneMinutePulse THEN
       #rTemp := #rQuality * 100.0;
       #diQuality := ROUND(#rTemp);
       "fcMQTT_dint"(sInTopic := 'iot-2/evt/status/fmt/json',
                     iInQoS := 1,
                     sInValueFormat := '{"d":{"Quality":<<value>>}}',
                     diInValue := #diQuality);
   END_IF;
END_REGION

REGION Network 8: Calculate OEE
   // OEE = Availability * Performance * Quality
   RUNG wire#powerrail
      Mul(in1 := #rAvailability, in2 := #rPerformance, in3 := #rQuality, out => #rOEE)
   END_RUNG
   RUNG wire#powerrail
      Contact( #bOneMinutePulse )
      Mul(in1 := #rOEE, in2 := 100.0, out => #rTemp)
      { S7_Templates := "[SrcType := Real, DestType := DInt]" } Round(in := #rTemp, out => #diOEE_Per)
      "fcMQTT_dint"(sInTopic := 'iot-2/evt/status/fmt/json', iInQoS := 1, sInValueFormat := '{"d":{"OEE":<<value>>}}', diInValue := #diOEE_Per)
   END_RUNG
   RUNG wire#powerrail
      Contact( #bOneMinutePulse )
      #AVG_OEE(rInValue := #rOEE, iInBufferSize := 10, rOutAverage => #rTemp, rOutMin =>, rOutMax =>, iOutBufferSize =>, bOutError =>)
      Mul(in1 := #rTemp, in2 := 100.0, out => #rTemp)
      { S7_Templates := "[SrcType := Real, DestType := DInt]" } Round(in := #rTemp, out => #diOEE_PerAvg)
      "fcMQTT_dint"(sInTopic := 'iot-2/evt/status/fmt/json', iInQoS := 1, sInValueFormat := '{"d":{"OEE_Avg":<<value>>}}', diInValue := #diOEE_PerAvg)
   END_RUNG
   // the same network as SCL:
   #rOEE := #rAvailability * #rPerformance * #rQuality;
   IF #bOneMinutePulse THEN
       #rTemp := #rOEE * 100.0;
       #diOEE_Per := ROUND(#rTemp);
       "fcMQTT_dint"(sInTopic := 'iot-2/evt/status/fmt/json',
                     iInQoS := 1,
                     sInValueFormat := '{"d":{"OEE":<<value>>}}',
                     diInValue := #diOEE_Per);
   END_IF;
   #AVG_OEE(EN := #bOneMinutePulse, rInValue := #rOEE, iInBufferSize := 10, rOutAverage => #rTemp, ENO => #_w1);   // "fbRunningAverage"
   IF #_w1 THEN
       #rTemp := #rTemp * 100.0;
       #diOEE_PerAvg := ROUND(#rTemp);
       "fcMQTT_dint"(sInTopic := 'iot-2/evt/status/fmt/json',
                     iInQoS := 1,
                     sInValueFormat := '{"d":{"OEE_Avg":<<value>>}}',
                     diInValue := #diOEE_PerAvg);
   END_IF;
END_REGION

REGION Network 9: Machine runtime timer (seconds per minute)
   #TONR_MachineRunTime(IN := #bMachineRunning, R := #bOneMinutePulse, PT := t#1m);   // TONR
END_REGION

REGION Network 10: Reset minute counters
   RUNG wire#powerrail
      Contact( #bOneMinutePulse )
      Move(in := 0, out1 => #diPartsBadMinute)
      Move(in := 0, out1 => #diPartsGoodMinute)
   END_RUNG
   // the same network as SCL:
   IF #bOneMinutePulse THEN
       #diPartsBadMinute := 0;
       #diPartsGoodMinute := 0;
   END_IF;
END_REGION

REGION Network 11: Send periodic message
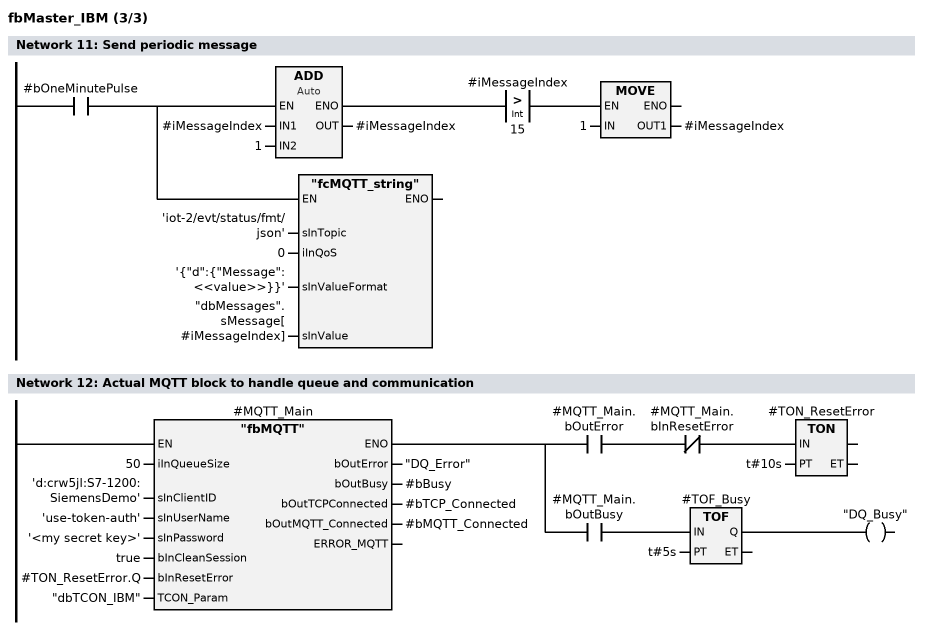
   RUNG wire#powerrail
      Contact( #bOneMinutePulse )
      wire#w1
      Add(in1 := #iMessageIndex, in2 := 1, out => #iMessageIndex)
      { S7_Templates := "SrcType := Int" } GT_Contact(in1 := #iMessageIndex, in2 := 15)
      Move(in := 1, out1 => #iMessageIndex)
   END_RUNG
   RUNG wire#w1
      "fcMQTT_string"(sInTopic := 'iot-2/evt/status/fmt/json', iInQoS := 0, sInValueFormat := '{"d":{"Message":<<value>>}}', sInValue := "dbMessages".sMessage[#iMessageIndex])
   END_RUNG
   // the same network as SCL:
   IF #bOneMinutePulse THEN #iMessageIndex := #iMessageIndex + 1; END_IF;
   IF #bOneMinutePulse AND (#iMessageIndex > 15) THEN #iMessageIndex := 1; END_IF;
   IF #bOneMinutePulse THEN
       "fcMQTT_string"(sInTopic := 'iot-2/evt/status/fmt/json',
                       iInQoS := 0,
                       sInValueFormat := '{"d":{"Message":<<value>>}}',
                       sInValue := "dbMessages".sMessage[#iMessageIndex]);
   END_IF;
END_REGION

REGION Network 12: Actual MQTT block to handle queue and communication
   #MQTT_Main(iInQueueSize := 50,   // "fbMQTT"
              sInClientID := 'd:crw5jl:S7-1200:SiemensDemo',
              sInUserName := 'use-token-auth',
              sInPassword := '<my secret key>',
              bInCleanSession := true,
              bInResetError := #TON_ResetError.Q,
              TCON_Param := "dbTCON_IBM",
              bOutError => "DQ_Error",
              bOutBusy => #bBusy,
              bOutTCPConnected => #bTCP_Connected,
              bOutMQTT_Connected => #bMQTT_Connected,
              ENO => #_w1);
   #TON_ResetError(IN := #_w1 AND #MQTT_Main.bOutError AND NOT #MQTT_Main.bInResetError, PT := t#10s);   // TON
   #TOF_Busy(IN := #_w1 AND #MQTT_Main.bOutBusy, PT := t#5s);   // TOF
   "DQ_Busy" := #TOF_Busy.Q;
END_REGION
END_FUNCTION_BLOCK

FUNCTION "fcMQTT_dint" : Void   // FC1, SCL
{ S7_Optimized_Access := 'TRUE' }
VERSION : 0.1
   VAR_INPUT
      sInTopic : String;   // MQTT topic to publish
      iInQoS : Int;   // QoS integer value (0-2)
      sInValueFormat : String;   // JSON format string. Format should have <<value>>, it will be replaced with actual value parameter
      diInValue : DInt;   // Actual value
   END_VAR
   VAR_TEMP
      iPos : Int;
      sValue : String;
      sTemp : String;
   END_VAR
BEGIN
   // Generate new global index to write    
   "dbMQTT_Queue".iIndexWrite := "dbMQTT_Queue".iIndexWrite + 1;
   // Check queue index at the end of the queue
   IF ("dbMQTT_Queue".iIndexWrite > "dbMQTT_Queue".iIndexMax) OR ("dbMQTT_Queue".iIndexWrite <=0) THEN
       "dbMQTT_Queue".iIndexWrite := 1;
   END_IF;

   IF "dbMQTT_Queue".Element["dbMQTT_Queue".iIndexWrite].iStatus <> 0 THEN
       // Queue overfill detected
       "dbMQTT_Queue".bErrorOverfill := true;
   END_IF;

   // Assing element to the queue
   // TODO: BLKMOV instead?
   "dbMQTT_Queue".Element["dbMQTT_Queue".iIndexWrite].sTopic := #sInTopic;
   "dbMQTT_Queue".Element["dbMQTT_Queue".iIndexWrite].iQOS := #iInQoS;
   #sValue := S_CONV(IN := #diInValue);
   IF #diInValue >= 0 THEN
       // Remove + sign from the string
       #sValue := DELETE(IN := #sValue, L := 1, P := 1);
   END_IF;

   // Replace JSON string if needed
   #iPos := FIND(IN1 := #sInValueFormat, IN2 := '<<value>>');
   IF (LEN(IN := #sInValueFormat) = 0) OR (#iPos <= 0) THEN
       "dbMQTT_Queue".Element["dbMQTT_Queue".iIndexWrite].sValue := #sValue;
   ELSE
       #sTemp := DELETE(IN := #sInValueFormat, L := 9, P := #iPos);
       "dbMQTT_Queue".Element["dbMQTT_Queue".iIndexWrite].sValue := INSERT(IN1 := #sTemp, IN2 := #sValue, P := #iPos-1);
   END_IF;

   // Update MQTT status
   "dbMQTT_Queue".Element["dbMQTT_Queue".iIndexWrite].iStatus := 10;

   ENO := TRUE;
END_FUNCTION

FUNCTION "fcMQTT_string" : Void   // FC2, SCL
{ S7_Optimized_Access := 'TRUE' }
VERSION : 0.1
   VAR_INPUT
      sInTopic : String;   // MQTT topic to publish
      iInQoS : Int;   // QoS integer value (0-2)
      sInValueFormat : String;   // JSON format string. Format should have <<value>>, it will be replaced with actual value parameter
      sInValue : String;   // Actual value
   END_VAR
   VAR_TEMP
      iPos : Int;
      sTemp : String;
   END_VAR
BEGIN
   // Generate new global index to write    
   "dbMQTT_Queue".iIndexWrite := "dbMQTT_Queue".iIndexWrite + 1;
   // Check queue index at the end of the queue
   IF ("dbMQTT_Queue".iIndexWrite > "dbMQTT_Queue".iIndexMax) OR ("dbMQTT_Queue".iIndexWrite <=0) THEN
       "dbMQTT_Queue".iIndexWrite := 1;
   END_IF;

   IF "dbMQTT_Queue".Element["dbMQTT_Queue".iIndexWrite].iStatus <> 0 THEN
       // Queue overfill detected
       "dbMQTT_Queue".bErrorOverfill := true;
   END_IF;

   // TODO: BLKMOV instead?
   "dbMQTT_Queue".Element["dbMQTT_Queue".iIndexWrite].sTopic := #sInTopic;
   "dbMQTT_Queue".Element["dbMQTT_Queue".iIndexWrite].iQOS := #iInQoS;

   // Replace JSON string if needed
   #iPos := FIND(IN1 := #sInValueFormat, IN2 := '<<value>>');
   IF (LEN(IN := #sInValueFormat) = 0) OR (#iPos <= 0) THEN
       "dbMQTT_Queue".Element["dbMQTT_Queue".iIndexWrite].sValue := #sInValue;
   ELSE
       #sTemp := DELETE(IN := #sInValueFormat, L := 9, P := #iPos);
       "dbMQTT_Queue".Element["dbMQTT_Queue".iIndexWrite].sValue := INSERT(IN1 := #sTemp, IN2 := #sInValue, P := #iPos-1);
   END_IF;

   "dbMQTT_Queue".Element["dbMQTT_Queue".iIndexWrite].iStatus := 10;

   ENO := TRUE;
END_FUNCTION

ORGANIZATION_BLOCK "Main"   // OB1, LAD, ProgramCycle
TITLE = "Main Program Sweep (Cycle)"
{ S7_Optimized_Access := 'TRUE' }
VERSION : 0.1
   VAR_TEMP
      bTemp : Bool;
   END_VAR
BEGIN

REGION Network 1: Call master block (Adafruit)
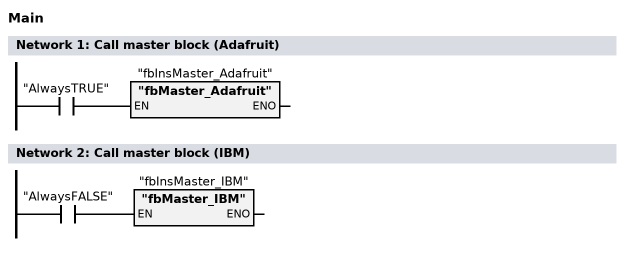
   RUNG wire#powerrail
      Contact( "AlwaysTRUE" )
      "fbInsMaster_Adafruit"()
   END_RUNG
   // the same network as SCL:
   IF "AlwaysTRUE" THEN
       "fbInsMaster_Adafruit"();   // "fbMaster_Adafruit"
   END_IF;
END_REGION

REGION Network 2: Call master block (IBM)
   RUNG wire#powerrail
      Contact( "AlwaysFALSE" )
      "fbInsMaster_IBM"()
   END_RUNG
   // the same network as SCL:
   IF "AlwaysFALSE" THEN
       "fbInsMaster_IBM"();   // "fbMaster_IBM"
   END_IF;
END_REGION
END_ORGANIZATION_BLOCK

// ===== library types =====

// folder: Errors

TYPE "udtError_Recipe"
AUTHOR : DMC
FAMILY : Error
VERSION : 0.1
   STRUCT
      ReportHeaderTimeOut : Bool;   // Save report header timed out, check database connection
      ReportFooterTimeOut : Bool;   // Save report footer timed out, check database connection
      ReportCommandsOverfill : Bool;   // Commands array overfilled, check database connection
      RepAppFailed : Bool;   // Reporting application connection failed
   END_STRUCT;
END_TYPE

// folder: Process

TYPE "udtRecipe"
AUTHOR : DMC
FAMILY : Recipe
VERSION : 0.0
   STRUCT
      sName : String[20];   // Recipe name
      sDescription : String[30];   // Recipe description
      iRecipe_ID : Int;   // Recipe ID
      iStatus : Int;   // Recipe loading status
      iBatchesToMake : Int;   // How many batches to make
      iBatchesMade : Int;   // How many batches already made
      iBatchesStarted : Int;   // How many batches started
      rMixerTemp : Real;   // Mixer temperature setpoint
      "Step" : Array[1..20] of Struct
         Command : Array[1..4] of Struct
            iCode : Int;   // Command code
            sName : String[30];   // Command name from commands array for HMI
            rSetpoint : Real;   // Command set point
            rFlowSP : Real;   // Flowrate setpoint
         END_STRUCT;
         Agitation : Struct
            iCode : Int;   // Agitation code
            sName : String[30];   // Agitation name from commands array for HMI
            rTime : Real;   // Agitation time (min)
         END_STRUCT;
      END_STRUCT;
   END_STRUCT;
END_TYPE

TYPE "udtRecipeCommand"
AUTHOR : DMC
FAMILY : Recipe
VERSION : 0.1
   STRUCT
      iStatus : Int;   // Command status
      iType : Int;   // 10-Automatic, 20-Manual
      bReady : Bool;   // Status ready bit
      sName : String[30];   // Command name
      sTime_Start : String[30];   // Time Command start
      sTime_Finish : String[30];   // Time Command finish
      rSetpoint : Real;   // Command set point
      rActual : Real;   // Command actual weight
      rPreact : Real;   // Preact
      rSlow_Preact : Real;   // Slow speed preact
      rTolerance : Real;   // Tolerance
      rTotal : Real;   // Total amount for recipe
      rFlowSP : Real;   // Flowrate setpoint
      rFlowActual : Real;   // Flowrate actual
      rTemperature : Real;   // Ingredient temperature
      rReportTimeDelay : Real;   // Save ingredient report every "delay" seconds
      rReportTimeActual : Real;   // Actual delay time
      iCommandStartStatus : Int;   // 0-disabled, 10-started, 20-start time saved
   END_STRUCT;
END_TYPE

TYPE "udtRecipeCommands"
AUTHOR : DMC
FAMILY : Recipe
VERSION : 0.1
   STRUCT
      Command : Array[1..100] of "udtRecipeCommand";
   END_STRUCT;
END_TYPE

TYPE "udtCurrentCommands"
AUTHOR : DMC
FAMILY : Recipe
VERSION : 0.1
   STRUCT
      Command : Array[1..4] of "udtRecipeCommand";
   END_STRUCT;
END_TYPE

TYPE "udtStdReportOperV2"
VERSION : 0.1
   STRUCT
      iBatchUID : Int;   // Batch unique identifier, generated on PLC side
      Header : "udtStdReportHeaderV2";
      Command : "udtStdReportCommandV2";
      Footer : "udtStdReportFooterV2";
      iReportingStatus : Int;   // Reporting status
   END_STRUCT;
END_TYPE

TYPE "udtStdReportHeaderV2"
VERSION : 0.1
   STRUCT
      iLineNo : Int;   // Line number
      iMixerNo : Int;   // Mixer number
      iStatus : Int;   // Batch status
      sName : String[30];   // Recipe name
      sDescription : String[30];   // Recipe description
      iRecipeID : Int;   // Recipe ID
      iBatchNumber : Int;   // Batch number
      sTimeStart : String[30];
      rMixerTemp : Real;   // Mixer temperature
   END_STRUCT;
END_TYPE

TYPE "udtStdReportCommandV2"
VERSION : 0.1
   STRUCT
      iStep : Int;   // Command step number
      iStatus : Int;   // Command status
      sName : String[30];   // Command name
      iCode : Int;   // Command code
      iIngredientType : Int;   // Command type
      sTimeStart : String[30];   // Time Command start
      sTimeFinish : String[30];   // Time Command finish
      rSetpoint : Real;   // Command set point
      rActual : Real;   // Command actual value
      rTemperature : Real;   // Ingredient temperature
   END_STRUCT;
END_TYPE

TYPE "udtStdReportFooterV2"
VERSION : 0.1
   STRUCT
      iStatus : Int;   // Report status
      rMixerTemp : Real;   // Mixer temperature
      sTimeFinish : String[30];
   END_STRUCT;
END_TYPE

FUNCTION_BLOCK "fbRecipe"   // FB600, SCL
TITLE = Recipe control
{ S7_Optimized_Access := 'FALSE' }
AUTHOR : Boris
VERSION : 3.2
// 2/9/07 - Changing reporting functionality.
//  5/10/07 - Batch Count Totalled over All Three Mixers, count increments at beginning of batch
//  6/14/07 - Report timeout if status not ciReportDisable and not ciReportSaved (BC)
//  6/10/09 - CRP - Added code for to use StdReports instead of Reports. Comment out old Report code
   VAR_INPUT
      iInMode : Int;   // Sysytem mode
      iInLineNumber : Int;   // Line number
      iInMixerNumber : Int;   // Mixer number, start from 1
      bInRecipeReset : Bool;   // Cancel batch / reset recipe
      bInRecipePause : Bool;   // Pause recepe
      bInStepPause : Bool;   // Pause step
      bInStepSkip : Bool;   // skip curren step and jump to the next
      bInResetError : Bool;   // Reset Error
      rInMixerTemperature : Real;   // Mixer temperature
   END_VAR
   VAR_OUTPUT
      iOutRecipeStep : Int;   // Current recipe step
      iOutBatchNumber : Int;   // Current Batch Number
      iOutSequenceStep : Int;   // Internal sequence step number
      bOutStepNotReady : Bool;   // Step Not Ready
      bOutRecipeRunning : Bool;   // Recipe Running
      bOutStepPaused : Bool;   // Step Paused
      bOutError : Bool;   // Error Present
      ERROR_Recipe : "udtError_Recipe";
   END_VAR
   VAR_IN_OUT
      rMixerTemp_SP : Real;   // Mixer temperature setpoint
      RecipeMaster : "udtRecipe";   // recipe downloaded from database
      RecipeCurrent : "udtRecipe";   // currently running recipe
      Commands : "udtRecipeCommands";   // Recipe command
      CommandsCurrent : "udtCurrentCommands";   // Currently acive command
      AgitationCurrent : "udtRecipeCommand";   // Current agitation command
   END_VAR
   VAR
      iSEQUENCE_STEP : Int;   // Internal sequence step
      iRECIPE_STEP : Int;   // Recipe current step
      iBATCH_COUNTER : Int;   // Batch counter
      TON_RepAppTimeOut : TON_TIME;   // Reporting application failed (CurrentTime not changing)
      iReportFailCount : Int;   // Report timed out counter
      TON_1sec : TON_TIME;   // 1 second pulse timer
      sPrev_DateTime : String[30];   // Stored date time (updated from reporting application)
      CurReportOper : "udtStdReportOperV2";   // Current report operatio/header/status
      sTemp : String[30];
      sTempName : String[30];
      sTempStartTime : String[30];
      sTempEndTime : String[30];
      sTempDescription : String[30];
      sTempRecipeName : String[20];
      iTempID : Int;
      bTON_1sec : Bool;
   END_VAR
   VAR_TEMP
      I : Int;
      J : Int;
      iTemp : Int;
      iStatus : Int;
      bStepDone : Bool;   // Step Done
      bStepNotEmpty : Bool;   // Step Not Empty
      bRecipeRunning : Bool;   // Recipe is running
      bAllIngrReady : Bool;   // All ingredients are running
      bTimeNotChanged : Bool;   // Time not changed
      bTemp : Bool;   // temp variable
      sPrevDay : String[30];
      sNewDay : String[30];
   END_VAR
   VAR CONSTANT
      ciNUM_Commands : Int := 100;   // Commands array
      ciNUM_STEPS : Int := 20;   // Steps in recipe
      ciNUM_ING_PER_STEP : Int := 4;   // Ingredients per step
      ciNUM_Report_Commands : Int := 100;   // Commands in report array
      ciRECIPE_READY : Int;   // Recipe Ready
      ciRECIPE_NAMES_UPDATED : Int := 10;   // Recipe Names Updated
      ciRECIPE_CALC_TOTAL : Int := 15;   // Calculating total weight
      ciRECIPE_NEW : Int := 20;   // New Recipe
      ciRECIPE_RUNNING : Int := 30;   // Recipe Running
      ciIngredientAuto : Int := 10;   // Ingredient auto addition
      ciIngredientManual : Int := 20;   // Ingredeint manual addition
      ciIngredientBarrel : Int := 21;
      ciReportDisable : Int;   // Not ready
      ciReportReady : Int := 10;   // Ready to save to database
      ciReportSavingToDataBase : Int := 20;   // Saving in progress
      ciReportFailed : Int := 30;   // Saving failed
      ciReportSaved : Int := 40;   // Saved
      ciRESET : Int;   // Reset Reset
      ciRECIPE_STARTED : Int := 10;   // Recipe Started
      ciNEW_STEP : Int := 50;   // New Step
      ciSTEP_STARTED : Int := 60;   // Step Started
      ciWAIT_READY : Int := 62;   // Wait for Ingredient Ready
      ciWAIT_FOR_STEP_FINISHED : Int := 65;   // Wait for Step Finished
      ciSTEP_FINISHED : Int := 70;   // Step Finished
      ciSEQUENCE_FINISHED_OK : Int := 100;   // Sequence Finished OK
      ciSAVE_Report : Int := 110;   // Saving Report
   END_VAR
BEGIN


   IF #bInResetError THEN // Clear errors
       #ERROR_Recipe.ReportHeaderTimeOut := false;
       #ERROR_Recipe.ReportFooterTimeOut := false;    
       #ERROR_Recipe.ReportCommandsOverfill := false;
       #ERROR_Recipe.RepAppFailed := false;
   END_IF;    

   #TON_1sec (IN := NOT #bTON_1sec, PT := T#1S);

   //**********************************************************************************************************************
   // Ingredients Reporting block, bStepDone use in other steps
   #bStepDone := TRUE;
   FOR #I := 1 TO #ciNUM_Commands BY 1 DO    // Scan commands array
       #iStatus := #Commands.Command[#I].iStatus; // Use iStatus variable in this loop, for better speed.

       IF (#iStatus <> "IngredientStatus.Disable") AND (#iStatus <>"IngredientStatus.DoneReported") THEN    // if command enabled and not reported
           #bStepDone := FALSE; // Setp not disabled and not reported

           // Recipe canceled
           IF #bInRecipeReset THEN    // If reseting recipe - set status to canceled
               #iStatus := "IngredientStatus.RecipeCanceled";   // Overwrite status    
               #Commands.Command[#I].iStatus := #iStatus; // Save ingredeint status     
           END_IF;

           // Skip step button pressed
           IF (#iInMode="Modes.Auto") AND #bInStepPause AND #bInStepSkip THEN   // If skip step button pressed
               #iStatus := "IngredientStatus.StepCanceled";   // Overwrite status    
               #Commands.Command[#I].iStatus := #iStatus; // Save ingredeint status     
               //Report.Footer.iStatus := dbGlobals.IngredientStatus.StepCanceled;

               // STANDARD REPORTS. Update report status, status 120 - step canceled
               "fcStdReportBatchStatus" (
                                         iInLineNo := #iInLineNumber,    
                                         iInMixerNo := #iInMixerNumber,
                                         iInBatchStatus := 120, 
                                         MixerReportOperation := #CurReportOper
                                       );
               // STANDARD REPORTS. 


           END_IF;                


           // Ingredient started, save start time
           IF (#Commands.Command[#I].iCommandStartStatus = "CommandStartStatus.Started") THEN
               #Commands.Command[#I].sTime_Start := "dbGlobals".sCurrent_DateTime;
               #Commands.Command[#I].iCommandStartStatus := "CommandStartStatus.StartedTimeSaved";
               #Commands.Command[#I].rReportTimeActual := 0.0;   // Command started - reset reporting timer
           END_IF;    

           // Ingredient delivering, update interval timer
           IF (#iStatus = "IngredientStatus.DeliveringAuto") OR (#iStatus ="IngredientStatus.DeliveringAutoFast")
               OR (#iStatus = "IngredientStatus.DeliveringAutoSlow") OR (#iStatus ="IngredientStatus.DeliveringAutoTimeout") THEN    // Save intermediate report even in case of timeout!
               IF #Commands.Command[#I].rReportTimeDelay > 0.0 THEN // Update ingredint if report delay > 0 
                   IF #bTON_1sec THEN
                        // BC. Theoreticaly we have to add 0.01666666 to actual time (1minute/60pulses). But actualy timer is not exacly 1 sec, it seems like timer gets delay due to unknown reason
                        // BC. Instead of theoretical constant we using value calculated on current PLC over extended period of time (2min/105pulses=0.019047619047619047619047619047619).
                        #Commands.Command[#I].rReportTimeActual := #Commands.Command[#I].rReportTimeActual + 0.01904762;
                   END_IF;

                   IF  #Commands.Command[#I].rReportTimeActual >= #Commands.Command[#I].rReportTimeDelay THEN 
                       #iStatus := "IngredientStatus.IntermStatus"; // Overwrite local status, not in commands array
                       #Commands.Command[#I].rReportTimeActual := 0.0;
                   END_IF;
               ELSE 
                   #Commands.Command[#I].rReportTimeDelay := 0.0;
               END_IF;
           END_IF;

           // Ingredient done, save report to DB
           IF (#iStatus = "IngredientStatus.DoneOk") OR (#iStatus ="IngredientStatus.DoneTolError")
               OR (#iStatus = "IngredientStatus.Bypassed") OR (#iStatus ="IngredientStatus.StepCanceled") OR (#iStatus ="IngredientStatus.RecipeCanceled")
               OR (#iStatus = "IngredientStatus.IntermStatus") THEN   // Save command Report

               //Increase the report command index
   //            IF (Report.iCommandIndex > 0) AND (Report.iCommandIndex < ciNUM_Commands) THEN 
   //                Report.iCommandIndex := Report.iCommandIndex + 1;
   //            ELSE
   //                Report.iCommandIndex := 1;
   //            END_IF;  
   //          
   //            IF (Report.COMMAND[Report.iCommandIndex].iReportingStatus <> ciReportDisable) AND (Report.COMMAND[Report.iCommandIndex].iReportingStatus <> ciReportSaved) THEN
   //                ERROR_Recipe.ReportCommandsOverfill := true;
   //            END_IF;

               //Set Copy values to Report datablock
   //            Report.COMMAND[Report.iCommandIndex].iSTEP := iRECIPE_STEP;
   //            Report.COMMAND[Report.iCommandIndex].iSTATUS := iStatus;
   //            iTemp := BLKMOV (DSTBLK := Report.COMMAND[Report.iCommandIndex].sNAME, SRCBLK := Commands.COMMAND[I].sNAME);
   //            Report.COMMAND[Report.iCommandIndex].iCODE := I;
   //            Report.COMMAND[Report.iCommandIndex].iIngredientType := Commands.COMMAND[I].iType;
   //            iTemp := BLKMOV (DSTBLK := Commands.COMMAND[I].sTIME_FINISH, SRCBLK := dbGlobals.sCurrent_DateTime);    // Save command finish time
   //            iTemp := BLKMOV (DSTBLK := Report.COMMAND[Report.iCommandIndex].sTIME_START, SRCBLK := Commands.COMMAND[I].sTIME_START);
   //            iTemp := BLKMOV (DSTBLK := Report.COMMAND[Report.iCommandIndex].sTIME_FINISH, SRCBLK := Commands.COMMAND[I].sTIME_FINISH);
   //            Report.COMMAND[Report.iCommandIndex].rSETPOINT := Commands.COMMAND[I].rSETPOINT;
   //            Report.COMMAND[Report.iCommandIndex].rACTUAL := Commands.COMMAND[I].rACTUAL;
   //            Report.COMMAND[Report.iCommandIndex].rTemperature := Commands.COMMAND[I].rTemperature;

               //Update Command Finish time and save report
               #Commands.Command[#I].sTime_Finish := "dbGlobals".sCurrent_DateTime;    // Save command finish time

               #iTemp := BLKMOV(DSTBLK => #sTemp, SRCBLK := #Commands.Command[#I].sName);
               #iTemp := BLKMOV(DSTBLK => #sTempName, SRCBLK := #Commands.Command[#I].sName);
               #iTemp := BLKMOV(DSTBLK => #sTempStartTime, SRCBLK := #Commands.Command[#I].sTime_Start);
               #iTemp := BLKMOV(DSTBLK => #sTempEndTime, SRCBLK := #Commands.Command[#I].sTime_Finish);

               // STANDARD REPORTS. Save command into standard report.
               #bTemp := "fcStdReportOper" (
                                           iInLineNo := #iInLineNumber, 
                                           iInMixerNo := #iInMixerNumber,
                                           iInStepNumber := #iRECIPE_STEP,
                                           iInCommandStatus := #iStatus,
                                           sInCommandName := #sTemp,
                                           iInCommandCode := #I,
                                           iInCommandIngredientType := #Commands.Command[#I].iType,
                                           sInCommandTimeStart := #sTempStartTime,// sTempStartTime,// Commands.Command[I].sTIME_START,
                                           sInCommandTimeFinish := #sTempEndTime, //Commands.Command[I].sTIME_FINISH,
                                           rInCommandSetpoint :=#Commands.Command[#I].rSetpoint, //Commands.Command[I].rSETPOINT,
                                           rInCommandActual := #Commands.Command[#I].rActual,
                                           rInCommandTemperature := #Commands.Command[#I].rTemperature,
                                           MixerReportOperation := #CurReportOper
                                       );
                IF (#bTemp = false) THEN
                   #ERROR_Recipe.ReportCommandsOverfill := true;
                END_IF;
                // STANDARD REPORTS.



                IF (#iStatus <> "IngredientStatus.IntermStatus") THEN    // Do not change ingredient status if save intermediate step
                    #Commands.Command[#I].iStatus := "IngredientStatus.DoneReported"; // Update command status to reported
                   #Commands.Command[#I].iCommandStartStatus := "CommandStartStatus.Disable";    // If command reported - reset start time status              
               END_IF;
              // Report.COMMAND[Report.iCommandIndex].iReportingStatus := ciReportReady;  // Update report command status
           END_IF;            
       END_IF;

   END_FOR;

   IF #bInRecipeReset THEN    // If recipe reset - save Report
       IF (#iSEQUENCE_STEP<>#ciRESET) THEN    // Recipe in progress, save report footer
           //Report.Footer.iStatus := dbGlobals.IngredientStatus.RecipeCanceled;
           #iSEQUENCE_STEP := #ciSTEP_FINISHED;
           #iRECIPE_STEP := #ciNUM_STEPS;    // Set current Step to last step in sequence
       ELSE 
           #iRECIPE_STEP := 0;    // Recipe not started yet, reset recipe steps
       END_IF;   

       // STANDARD REPORTS. Update report status, status 130 - recipe canceled
       "fcStdReportBatchStatus" (
                                iInLineNo := #iInLineNumber, 
                                iInMixerNo := #iInMixerNumber,
                                iInBatchStatus := 130,
                                MixerReportOperation := #CurReportOper
                              );
       // STANDARD REPORTS. 


   END_IF;

   //**********************************************************************************************************************
   IF #RecipeMaster.iStatus = #ciRECIPE_NEW THEN // New recipe has been downloaded
       FOR #I := 1 TO #ciNUM_STEPS BY 1 DO   // Populate recipe command names from Commands array
           FOR #J := 1 TO #ciNUM_ING_PER_STEP BY 1 DO
               #iTemp := BLKMOV (DSTBLK => #RecipeMaster."Step"[#I].Command[#J].sName, SRCBLK := #Commands.Command[#RecipeMaster."Step"[#I].Command[#J].iCode].sName);
           END_FOR;
               #iTemp := BLKMOV (DSTBLK => #RecipeMaster."Step"[#I].Agitation.sName, SRCBLK := #Commands.Command[#RecipeMaster."Step"[#I].Agitation.iCode].sName);
       END_FOR;
       #RecipeMaster.iStatus := #ciRECIPE_NAMES_UPDATED;


   END_IF;

   //**********************************************************************************************************************

   #bRecipeRunning := true;     // Recipe running
   #bOutStepPaused := false;    // Assume step not paused
   CASE #iSEQUENCE_STEP OF
   //**********************************************************************************************************************
       #ciRESET                                     : // Copy Master recipe to Current recipe
           IF  (#RecipeMaster.iStatus = #ciRECIPE_CALC_TOTAL) THEN // Total updated on all mixers
               #RecipeMaster.iStatus := #ciRECIPE_READY;      
           END_IF;

           IF  (#RecipeCurrent.iStatus = #ciRECIPE_READY) AND (#RecipeMaster.iStatus=#ciRECIPE_NAMES_UPDATED) THEN // If recipe names has been updated
                   #iTemp := BLKMOV (DSTBLK => #RecipeCurrent, SRCBLK := #RecipeMaster);    // Copy new recipe
                   #RecipeMaster.iStatus := #ciRECIPE_CALC_TOTAL;      

           END_IF;

           IF (#RecipeMaster.iStatus = #ciRECIPE_CALC_TOTAL) THEN // Calculate total weight for each mixer
               #iBATCH_COUNTER := 0;    // Reset mixer batch number for each mixer

               #rMixerTemp_SP := #RecipeCurrent.rMixerTemp;  // Set the mixer temp from recipe only when new recipe is downloaded
               FOR #I := 1 TO #ciNUM_Commands BY 1 DO    // Reset total weight
                   #Commands.Command[#I].rTotal := 0.0;    
               END_FOR;
               FOR #I := 1 TO #ciNUM_STEPS BY 1 DO   // Calculate total weight
                   FOR #J := 1 TO #ciNUM_ING_PER_STEP BY 1 DO
                       IF #RecipeCurrent."Step"[#I].Command[#J].iCode > 0 THEN 
                           #Commands.Command[#RecipeCurrent."Step"[#I].Command[#J].iCode].rTotal := #Commands.Command[#RecipeCurrent."Step"[#I].Command[#J].iCode].rTotal + #RecipeCurrent."Step"[#I].Command[#J].rSetpoint;                
                       END_IF;
                   END_FOR;
               END_FOR;
           END_IF;

           IF (#iInMode="Modes.Auto") AND (#RecipeMaster.iStatus=#ciRECIPE_READY) AND NOT #bInRecipePause AND (#RecipeCurrent.iBatchesMade <= #RecipeCurrent.iBatchesToMake) THEN // If in Auto mode and start recipe input and batches counter OK
               #iSEQUENCE_STEP                   := #ciRECIPE_STARTED; // Jump to the next step
           ELSE     
               #iRECIPE_STEP                     := 0; // Set step 0 to indicate end of sequence
           END_IF;
           #bRecipeRunning := false;    // Recipe not running

   //**********************************************************************************************************************
       #ciRECIPE_STARTED                            : // Clear setpoints, load all ingridients setpoints of all steps for test
           FOR #I := 1 TO #ciNUM_Commands BY 1 DO
               #Commands.Command[#I].iStatus           := "IngredientStatus.Disable";
               #Commands.Command[#I].rSetpoint         := 0.0;    
               #Commands.Command[#I].rTotal            := 0.0;    
               #Commands.Command[#I].rActual           := 0.0;
               #Commands.Command[#I].sTime_Start := "sEmpty";
               #Commands.Command[#I].sTime_Finish := "sEmpty";
               #Commands.Command[#I].rReportTimeActual   := 0.0;    
               #Commands.Command[#I].iCommandStartStatus := "CommandStartStatus.Disable";
           END_FOR;

           #iBATCH_COUNTER  := #RecipeCurrent.iBatchesStarted + 1;               // Increment mixer batch number (global per mixer)
           #RecipeCurrent.iBatchesStarted := #RecipeCurrent.iBatchesStarted + 1;  // Increment recipe batch number (global per recipe)

           FOR #I := 1 TO #ciNUM_STEPS BY 1 DO   // Calculate total weight
               FOR #J := 1 TO #ciNUM_ING_PER_STEP BY 1 DO
                   IF #RecipeCurrent."Step"[#I].Command[#J].iCode > 0 THEN 
                       #Commands.Command[#RecipeCurrent."Step"[#I].Command[#J].iCode].rTotal := #Commands.Command[#RecipeCurrent."Step"[#I].Command[#J].iCode].rTotal + #RecipeCurrent."Step"[#I].Command[#J].rSetpoint;                
                   END_IF;
               END_FOR;
           END_FOR;      

           // Update Report header
   //        iTemp := BLKMOV (DSTBLK := Report.Header.sNAME, SRCBLK := RecipeCurrent.sNAME);        
   //        Report.Header.iRECIPE_ID                := RecipeCurrent.iRECIPE_ID; 
   //        Report.Header.iBATCH_NUMBER             := iBATCH_COUNTER;    
   //        iTemp := BLKMOV (DSTBLK := Report.Header.sTIME_START, SRCBLK := dbGlobals.sCurrent_DateTime);
   //        Report.Header.rMIXER_TEMP               := rInMixerTemperature;        
   //        Report.Header.iReportingStatus          := ciReportReady;

           // Clear Report array
   //        FOR I := 1 TO ciNUM_Report_Commands BY 1 DO
   //            Report.COMMAND[I].iSTEP := 0;
   //            Report.COMMAND[I].iSTATUS := dbGlobals.IngredientStatus.DISABLE;
   //            iTemp := BLKMOV (DSTBLK := Report.COMMAND[I].sNAME, SRCBLK := dbGlobals.sEMPTY);
   //            Report.COMMAND[I].iCODE := 0;
   //            Report.COMMAND[I].iIngredientType := 0;
   //            iTemp := BLKMOV (DSTBLK := Report.COMMAND[I].sTIME_START, SRCBLK := dbGlobals.sEMPTY);
   //            iTemp := BLKMOV (DSTBLK := Report.COMMAND[I].sTIME_FINISH, SRCBLK := dbGlobals.sEMPTY);
   //            Report.COMMAND[I].rSETPOINT := 0.0;
   //            Report.COMMAND[I].rACTUAL := 0.0;
   //            Report.COMMAND[I].rTemperature := 0.0;
   //            Report.COMMAND[I].iReportingStatus := ciReportDisable;
   //        END_FOR;
   //        Report.iCommandIndex := 0;
   //        
   //        // Clear Report footer
   //        Report.Footer.iStatus := dbGlobals.IngredientStatus.DISABLE;
   //        Report.Footer.rMixer_Temp := 0.0;
   //        iTemp := BLKMOV (DSTBLK := Report.Footer.sTIME_FINISH, SRCBLK := dbGlobals.sEMPTY);
   //        Report.Footer.iReportingStatus := ciReportDisable;

   // STANDARD REPORTS. Call standard report function (batch start)
           #bTemp := "fcStdReportBatchStart" ( 
                                               iInLineNo := #iInLineNumber, 
                                               iInMixerNo := #iInMixerNumber,
                                               sInFormulaName :=  #sTempRecipeName, 
                                               sInFormulaDescription := #sTempDescription, //dbRecipes.Current[iInRecipeIndex].sDescription,
                                               iInFormulaID := #iTempID, //dbRecipes.Current[iInRecipeIndex].iRecipe_ID,
                                               iInBatchNumber := #iBATCH_COUNTER,
                                               sInTimeStart := "dbGlobals".sCurrent_DateTime,
                                               rInMixerTempStart := #rInMixerTemperature,
                                               MixerReportOperation := #CurReportOper
                                          );
           IF (#bTemp = false) THEN
               #ERROR_Recipe.ReportCommandsOverfill := true;
           END_IF;
           // STANDARD REPORTS.   



           #iRECIPE_STEP                             := 1;  // Set step number to indicate recipe start
           #iSEQUENCE_STEP                           := #ciNEW_STEP;

   //**********************************************************************************************************************
       #ciNEW_STEP                                  : // Load setpoints
           #bStepNotEmpty := false; // Be sure step is not empty
           FOR #I := 1 TO #ciNUM_ING_PER_STEP BY 1 DO    // Commands setpoints
               IF #RecipeCurrent."Step"[#iRECIPE_STEP].Command[#I].iCode > 0 THEN 
                   #Commands.Command[#RecipeCurrent."Step"[#iRECIPE_STEP].Command[#I].iCode].rSetpoint := #Commands.Command[#RecipeCurrent."Step"[#iRECIPE_STEP].Command[#I].iCode].rSetpoint + #RecipeCurrent."Step"[#iRECIPE_STEP].Command[#I].rSetpoint;
                   #Commands.Command[#RecipeCurrent."Step"[#iRECIPE_STEP].Command[#I].iCode].iStatus   := "IngredientStatus.Disable";
                   #bStepNotEmpty := true; 
               END_IF;
           END_FOR;
           IF #RecipeCurrent."Step"[#iRECIPE_STEP].Agitation.iCode > 0 THEN 
               #Commands.Command[#RecipeCurrent."Step"[#iRECIPE_STEP].Agitation.iCode].rSetpoint := #RecipeCurrent."Step"[#iRECIPE_STEP].Agitation.rTime;    // Copy agitation command
               #Commands.Command[#RecipeCurrent."Step"[#iRECIPE_STEP].Agitation.iCode].iStatus := "IngredientStatus.Disable";
               #bStepNotEmpty := true;
           END_IF;

           IF #bStepNotEmpty THEN 
               #iSEQUENCE_STEP := #ciSTEP_STARTED;
           ELSE
               #iSEQUENCE_STEP := #ciWAIT_FOR_STEP_FINISHED; // Current step empty jump to the next step
           END_IF;    

   //**********************************************************************************************************************
       #ciSTEP_STARTED                              : // Wait step unpaused
           #bOutStepPaused := true; // Seems like step paused
           IF (#iInMode="Modes.Auto") AND NOT #bInStepPause THEN    // Recipe not paused - enable Commands
               FOR #I := 1 TO #ciNUM_ING_PER_STEP BY 1 DO    // Commands setpoints
                   IF #RecipeCurrent."Step"[#iRECIPE_STEP].Command[#I].iCode > 0 THEN 
                       #Commands.Command[#RecipeCurrent."Step"[#iRECIPE_STEP].Command[#I].iCode].iStatus   := "IngredientStatus.NotReady";    // Set command status to NOT_READY, if subsystem is ready it will reset it to READY        
                   END_IF;
               END_FOR;
               IF #RecipeCurrent."Step"[#iRECIPE_STEP].Agitation.iCode > 0 THEN 
                   #Commands.Command[#RecipeCurrent."Step"[#iRECIPE_STEP].Agitation.iCode].iStatus := "IngredientStatus.NotReady";    // Set command status to NOT_READY, if subsystem is ready it will reset it to READY        
               END_IF;                       
               #iSEQUENCE_STEP := #ciWAIT_READY;
               #bOutStepPaused  := false;   // Step not paused any more
           END_IF;

           IF (#iInMode="Modes.Auto") AND #bInStepPause AND #bInStepSkip THEN   // If skip step button pressed
               FOR #I := 1 TO #ciNUM_ING_PER_STEP BY 1 DO    // Commands setpoints
                   IF #RecipeCurrent."Step"[#iRECIPE_STEP].Command[#I].iCode > 0 THEN 
                       #Commands.Command[#RecipeCurrent."Step"[#iRECIPE_STEP].Command[#I].iCode].iStatus := "IngredientStatus.StepCanceled";
                   END_IF;
               END_FOR;
               IF #RecipeCurrent."Step"[#iRECIPE_STEP].Agitation.iCode > 0 THEN 
                   #Commands.Command[#RecipeCurrent."Step"[#iRECIPE_STEP].Agitation.iCode].iStatus := "IngredientStatus.StepCanceled";
               END_IF;                       
               #iSEQUENCE_STEP := #ciWAIT_FOR_STEP_FINISHED;   // Jump to the next step
               #bOutStepPaused := false;    // Step not paused any more
             //  Report.Footer.iStatus := dbGlobals.IngredientStatus.StepCanceled;
           END_IF;

   //**********************************************************************************************************************
       #ciWAIT_READY                                : // Wait for all ingredients on current step to be ready
           #bAllIngrReady := true;  // Check respondes from all system READY
           FOR #I := 1 TO #ciNUM_ING_PER_STEP BY 1 DO    // Check Commands ready status

               IF (#RecipeCurrent."Step"[#iRECIPE_STEP].Command[#I].iCode > 0) AND (#Commands.Command[#RecipeCurrent."Step"[#iRECIPE_STEP].Command[#I].iCode].iStatus <> "IngredientStatus.Ready") THEN
                   #bAllIngrReady := false; // This system not ready
                   EXIT;
               END_IF;
           END_FOR;
           IF (#RecipeCurrent."Step"[#iRECIPE_STEP].Agitation.iCode > 0) AND (#Commands.Command[#RecipeCurrent."Step"[#iRECIPE_STEP].Agitation.iCode].iStatus <> "IngredientStatus.Ready") THEN
               #bAllIngrReady := false; // Agitation not ready
           END_IF;                       

           IF #bAllIngrReady THEN    // All systems are ready
               FOR #I := 1 TO #ciNUM_ING_PER_STEP BY 1 DO    // Commands setpoints
                   IF #RecipeCurrent."Step"[#iRECIPE_STEP].Command[#I].iCode > 0 THEN 
                       IF (#Commands.Command[#RecipeCurrent."Step"[#iRECIPE_STEP].Command[#I].iCode].iType = #ciIngredientManual OR #Commands.Command[#RecipeCurrent."Step"[#iRECIPE_STEP].Command[#I].iCode].iType = #ciIngredientBarrel) THEN 
                           #Commands.Command[#RecipeCurrent."Step"[#iRECIPE_STEP].Command[#I].iCode].iStatus := "IngredientStatus.EnableManual";   // Start manual Command
                       ELSE
                           #Commands.Command[#RecipeCurrent."Step"[#iRECIPE_STEP].Command[#I].iCode].iStatus := "IngredientStatus.EnableAuto";   // Start auto Command
                       END_IF;
                   END_IF;
               END_FOR;

               IF (#RecipeCurrent."Step"[#iRECIPE_STEP].Agitation.iCode > 0) THEN //Agitation steps
                   IF (#Commands.Command[#RecipeCurrent."Step"[#iRECIPE_STEP].Agitation.iCode].iType = #ciIngredientManual OR #Commands.Command[#RecipeCurrent."Step"[#iRECIPE_STEP].Command[#I].iCode].iType = #ciIngredientBarrel) THEN 
                       #Commands.Command[#RecipeCurrent."Step"[#iRECIPE_STEP].Agitation.iCode].iStatus := "IngredientStatus.EnableManual";
                   ELSE
                       #Commands.Command[#RecipeCurrent."Step"[#iRECIPE_STEP].Agitation.iCode].iStatus := "IngredientStatus.EnableAuto";
                   END_IF; 
               END_IF;    

               #iSEQUENCE_STEP                       := #ciWAIT_FOR_STEP_FINISHED;
           ELSE
               #iSEQUENCE_STEP                       := #ciWAIT_READY;
           END_IF;    

   //**********************************************************************************************************************
       #ciWAIT_FOR_STEP_FINISHED                    : // Wait for ingridients to be loaded, copy current ingredient status        
               IF #bStepDone THEN   // Step done bit from Report loop
                   #iSEQUENCE_STEP                       := #ciSTEP_FINISHED;
               ELSE;
                   #iSEQUENCE_STEP                       := #ciWAIT_FOR_STEP_FINISHED; // Wait on this step until all Commands done
               END_IF;

   //**********************************************************************************************************************                     
       #ciSTEP_FINISHED                             : // Step done: save Report, clear setpoints
           FOR #I := 1 TO #ciNUM_Commands BY 1 DO    // Clear Commands array
               #Commands.Command[#I].iStatus           := "IngredientStatus.Disable";
               #Commands.Command[#I].rSetpoint         := 0.0;    
               #Commands.Command[#I].rActual           := 0.0;
               #Commands.Command[#I].sTime_Start := "sEmpty";
               #Commands.Command[#I].sTime_Finish := "sEmpty";
               #Commands.Command[#I].rTemperature := 0.0;
               #Commands.Command[#I].rReportTimeActual := 0.0;
               #Commands.Command[#I].iCommandStartStatus := "CommandStartStatus.Disable";
           END_FOR;

           IF #iRECIPE_STEP < #ciNUM_STEPS THEN // if not last step, incriment step and start over
               #iRECIPE_STEP                        := #iRECIPE_STEP + 1;
               #iSEQUENCE_STEP                      := #ciNEW_STEP;
           ELSE        
               #iSEQUENCE_STEP                      := #ciSEQUENCE_FINISHED_OK;
           END_IF;   

   //**********************************************************************************************************************
       #ciSEQUENCE_FINISHED_OK                      :   // Recipe done OK
           #RecipeCurrent.iBatchesMade := #RecipeCurrent.iBatchesMade + 1;   // Increment made batches counter (global per recipe)

           // Set report footer status
           //IF (Report.Footer.iStatus = dbGlobals.IngredientStatus.Disable) THEN 
           //    Report.Footer.iStatus := dbGlobals.IngredientStatus.DoneOk;
           //END_IF;
           //Report.Footer.rMIXER_TEMP := rInMixerTemperature; // Update mixer temp
           //iTemp := BLKMOV (DSTBLK := Report.Footer.sTIME_FINISH, SRCBLK := dbGlobals.sCurrent_DateTime);
           //Report.Footer.iReportingStatus := ciReportReady;

           // STANDARD REPORTS. Update report status, Status 80 - recipe done ok
           #bTemp := "fcStdReportBatchComplete" (
                                                   iInLineNo := #iInLineNumber, 
                                                   iInMixerNo := #iInMixerNumber,
                                                   rInMixerTempFinish := #rInMixerTemperature, 
                                                   sInTimeFinish := "dbGlobals".sCurrent_DateTime,
                                                   iInBatchStatus  := 80,
                                                   MixerReportOperation := #CurReportOper
                                             );
           IF (#bTemp = false) THEN
               #ERROR_Recipe.ReportCommandsOverfill := true;
           END_IF;                                  
           // STANDARD REPORTS. 



           #iSEQUENCE_STEP := #ciSAVE_Report; // Save Report

   //**********************************************************************************************************************
       #ciSAVE_Report :   // Save Report - Spare step, not used any more
           #iSEQUENCE_STEP := #ciRESET; // Start Over
           #iRECIPE_STEP := 0; // Set step 0 to indicate end of sequence


       //    IF ((Report.Header.iReportingStatus = ciReportSaved) OR (Report.Header.iReportingStatus = ciReportFailed)) AND 
       //       ((Report.Footer.iReportingStatus = ciReportSaved) OR (Report.Footer.iReportingStatus = ciReportFailed)) THEN // report footer and header has been saved or failed
       //            iSEQUENCE_STEP := ciRESET; // Start Over
       //            iRECIPE_STEP := 0; // Set step 0 to indicate end of sequence                
       //    ELSE         
       //            iSEQUENCE_STEP := ciSAVE_Report; // Save Report
       //    END_IF;


   //**********************************************************************************************************************

   ELSE
       #iSEQUENCE_STEP                               := #ciRESET;
   END_CASE;

   //Report header timeout 
   //TON_ReportHeaderTimeOut (IN := (Report.Header.iReportingStatus <> ciReportDisable) AND (Report.Header.iReportingStatus <> ciReportSaved) AND (Report.Header.iReportingStatus <> ciReportFailed), PT := T#1M);/
   //IF TON_ReportHeaderTimeOut.Q THEN 
   //    Report.Header.iReportingStatus := ciReportFailed;
   //    ERROR_Recipe.ReportHeaderTimeOut := true;
   //END_IF;

   //Report Foooter Timeout    
   //TON_ReportFooterTimeOut (IN := (Report.Footer.iReportingStatus <> ciReportDisable) AND (Report.Footer.iReportingStatus <> ciReportSaved) AND (Report.Footer.iReportingStatus <> ciReportFailed), PT := T#1M);
   //IF TON_ReportFooterTimeOut.Q THEN 
   //    Report.Footer.iReportingStatus := ciReportFailed;    
   //    ERROR_Recipe.ReportFooterTimeOut := true;
   //END_IF;

   // Reporting screen communication error and batch number reset at the beginig of the day
   #bTimeNotChanged := ("dbGlobals".sCurrent_DateTime = #sPrev_DateTime);//EQ_STRNG (S1 := "dbGlobals".sCurrent_DateTime, S2 := #sPrev_DateTime); // Old string compare

   #TON_RepAppTimeOut (IN := #bTimeNotChanged AND NOT #ERROR_Recipe.RepAppFailed, PT := T#30S);
   IF #TON_RepAppTimeOut.Q THEN
       #ERROR_Recipe.RepAppFailed := true;        
   END_IF;    
   IF NOT #bTimeNotChanged THEN // Date/Time updated from reporting application
       #sPrevDay := MID(IN := #sPrev_DateTime, P := 9, L := 2);  // Read previous day number
       #sNewDay := MID(IN := "dbGlobals".sCurrent_DateTime, P := 9, L := 2);  // Read new day number    
       //IF NE_STRNG (S1 := sPrevDay, S2 := sNewDay) THEN   // Day number changed, reset batch counter for next batch
       //    iBATCH_COUNTER := 1;    // Reset batches counter (starts form 1);
       //END_IF;    
       #sPrev_DateTime := "dbGlobals".sCurrent_DateTime;   // Update previous time
   END_IF;    

   // Show active command and agitation on the screen
   FOR #I := 1 TO #ciNUM_ING_PER_STEP BY 1 DO    // Show active Commands on the screen
       IF (#iRECIPE_STEP <= #ciNUM_STEPS AND #iRECIPE_STEP > 0) THEN // JRM 20/27/2014 - added this so PLC did not throw PRG_FLT when iRECIPE_STEP = ciNUM_STEPS + 1
           IF (#RecipeCurrent."Step"[#iRECIPE_STEP].Command[#I].iCode > 0) THEN
               // tolerance error
               IF (#Commands.Command[#RecipeCurrent."Step"[#iRECIPE_STEP].Command[#I].iCode].iStatus = "IngredientStatus.DeliveringAutoTolError") THEN    // ingredient has tolerance error status
                   IF (#Commands.Command[#RecipeCurrent."Step"[#iRECIPE_STEP].Command[#I].iCode].rSetpoint < #CommandsCurrent.Command[#I].rSetpoint) THEN   // Setpoint on the HMI (current_comand) has been updated
                       #Commands.Command[#RecipeCurrent."Step"[#iRECIPE_STEP].Command[#I].iCode].rSetpoint := #CommandsCurrent.Command[#I].rSetpoint;    // update ingredient setpoint
                   END_IF;        
                   IF (#CommandsCurrent.Command[#I].iStatus = "IngredientStatus.UpdatedFromHMI") THEN   // Current command status has been update from HMI
                           #Commands.Command[#RecipeCurrent."Step"[#iRECIPE_STEP].Command[#I].iCode].iStatus := #CommandsCurrent.Command[#I].iStatus; // Update ingredient status
                   END_IF;               
               END_IF;

               // command bypassed
               IF (#Commands.Command[#RecipeCurrent."Step"[#iRECIPE_STEP].Command[#I].iCode].iStatus <> "IngredientStatus.Disable") AND
                   (#Commands.Command[#RecipeCurrent."Step"[#iRECIPE_STEP].Command[#I].iCode].iStatus <> "IngredientStatus.DoneReported") AND
                   (#CommandsCurrent.Command[#I].iStatus = "IngredientStatus.Bypassed") THEN
                   #Commands.Command[#RecipeCurrent."Step"[#iRECIPE_STEP].Command[#I].iCode].iStatus := "IngredientStatus.Bypassed"; // Bypass command
               END_IF;

               #iTemp := BLKMOV (DSTBLK => #CommandsCurrent.Command[#I], SRCBLK := #Commands.Command[#RecipeCurrent."Step"[#iRECIPE_STEP].Command[#I].iCode]);    // copy ingredient status to the HMI
               // overwrite current ingredient name from recipe, not from Commands array. Usefull to check recipe/ingredients consistency
               #iTemp := BLKMOV (DSTBLK => #CommandsCurrent.Command[#I].sName, SRCBLK := #RecipeCurrent."Step"[#iRECIPE_STEP].Command[#I].sName);
           ELSE
               #CommandsCurrent.Command[#I].iStatus           := "IngredientStatus.Disable";
               #CommandsCurrent.Command[#I].sName := "sEmpty";
               #CommandsCurrent.Command[#I].rSetpoint         := 0.0;    
               #CommandsCurrent.Command[#I].rActual           := 0.0;          
           END_IF;
       END_IF;
   END_FOR;

   //Agitation step
   IF (#iRECIPE_STEP <= #ciNUM_STEPS) THEN
       IF (#iRECIPE_STEP > 0) AND (#RecipeCurrent."Step"[#iRECIPE_STEP].Agitation.iCode > 0) THEN         
           #iTemp := BLKMOV (DSTBLK => #AgitationCurrent, SRCBLK := #Commands.Command[#RecipeCurrent."Step"[#iRECIPE_STEP].Agitation.iCode]);    // Show active agitation
       ELSE
           #AgitationCurrent.iStatus := "IngredientStatus.Disable";
           #AgitationCurrent.sName := "sEmpty";
           #AgitationCurrent.rSetpoint := 0.0;
           #AgitationCurrent.rActual := 0.0;                
       END_IF;
   END_IF;

   //IF (iInMixerNumber = 1) THEN  // If this is the first instance of the block
       #RecipeCurrent.iStatus := #ciRECIPE_READY;
   //END_IF;    
   IF (#RecipeCurrent.iStatus <> #ciRECIPE_RUNNING) AND #bRecipeRunning THEN // If recipe running
       #RecipeCurrent.iStatus := #ciRECIPE_RUNNING; // set run status
   END_IF;

   //Output recipe information    
   #iOutRecipeStep := #iRECIPE_STEP;
   #iOutBatchNumber := #iBATCH_COUNTER;
   #iOutSequenceStep := #iSEQUENCE_STEP;
   #bOutStepNotReady := (#iSEQUENCE_STEP = #ciWAIT_READY);
   #bOutRecipeRunning := #bRecipeRunning;
   #bOutError := #ERROR_Recipe.ReportHeaderTimeOut OR #ERROR_Recipe.ReportFooterTimeOut OR #ERROR_Recipe.ReportCommandsOverfill OR #ERROR_Recipe.RepAppFailed;

   ENO:=true;
END_FUNCTION_BLOCK

